// ---- DUTs/IO/Boxes/KL_65B88BEE.TcDUT
{attribute 'GeneratedUsingTerminal: KL1862-0001'}
{attribute addProperty BoxType "KL1862-0001"}
{attribute addProperty Description ""}
{attribute addProperty Physics ""}
{attribute addProperty Id "Channel_1AT %I*Channel_87C95E760Channel_2AT %I*Channel_87C95E760Channel_3AT %I*Channel_87C95E760Channel_4AT %I*Channel_87C95E760Channel_5AT %I*Channel_87C95E760Channel_6AT %I*Channel_87C95E760Channel_7AT %I*Channel_87C95E760Channel_8AT %I*Channel_87C95E760Channel_9AT %I*Channel_87C95E760Channel_10AT %I*Channel_87C95E760Channel_11AT %I*Channel_87C95E760Channel_12AT %I*Channel_87C95E760Channel_13AT %I*Channel_87C95E760Channel_14AT %I*Channel_87C95E760Channel_15AT %I*Channel_87C95E760Channel_16AT %I*Channel_87C95E760"}
{attribute addProperty CRC "1706593262"}
{attribute addProperty Size "0"}
TYPE KL_65B88BEE :
STRUCT
	{attribute addProperty Name "Channel_1"}
	Channel_1 : Channel_87C95E76;
	{attribute addProperty Name "Channel_2"}
	Channel_2 : Channel_87C95E76;
	{attribute addProperty Name "Channel_3"}
	Channel_3 : Channel_87C95E76;
	{attribute addProperty Name "Channel_4"}
	Channel_4 : Channel_87C95E76;
	{attribute addProperty Name "Channel_5"}
	Channel_5 : Channel_87C95E76;
	{attribute addProperty Name "Channel_6"}
	Channel_6 : Channel_87C95E76;
	{attribute addProperty Name "Channel_7"}
	Channel_7 : Channel_87C95E76;
	{attribute addProperty Name "Channel_8"}
	Channel_8 : Channel_87C95E76;
	{attribute addProperty Name "Channel_9"}
	Channel_9 : Channel_87C95E76;
	{attribute addProperty Name "Channel_10"}
	Channel_10 : Channel_87C95E76;
	{attribute addProperty Name "Channel_11"}
	Channel_11 : Channel_87C95E76;
	{attribute addProperty Name "Channel_12"}
	Channel_12 : Channel_87C95E76;
	{attribute addProperty Name "Channel_13"}
	Channel_13 : Channel_87C95E76;
	{attribute addProperty Name "Channel_14"}
	Channel_14 : Channel_87C95E76;
	{attribute addProperty Name "Channel_15"}
	Channel_15 : Channel_87C95E76;
	{attribute addProperty Name "Channel_16"}
	Channel_16 : Channel_87C95E76;
END_STRUCT
END_TYPE

// ---- DUTs/IO/Boxes/KL1872_65B88BEE.TcDUT
{attribute 'GeneratedUsingTerminal: KL1872'}
{attribute addProperty BoxType "KL1872"}
{attribute addProperty Description ""}
{attribute addProperty Physics ""}
{attribute addProperty Id "Channel_1AT %I*Channel_87C95E760Channel_2AT %I*Channel_87C95E760Channel_3AT %I*Channel_87C95E760Channel_4AT %I*Channel_87C95E760Channel_5AT %I*Channel_87C95E760Channel_6AT %I*Channel_87C95E760Channel_7AT %I*Channel_87C95E760Channel_8AT %I*Channel_87C95E760Channel_9AT %I*Channel_87C95E760Channel_10AT %I*Channel_87C95E760Channel_11AT %I*Channel_87C95E760Channel_12AT %I*Channel_87C95E760Channel_13AT %I*Channel_87C95E760Channel_14AT %I*Channel_87C95E760Channel_15AT %I*Channel_87C95E760Channel_16AT %I*Channel_87C95E760"}
{attribute addProperty CRC "1706593262"}
{attribute addProperty Size "0"}
TYPE KL1872_65B88BEE :
STRUCT
	{attribute addProperty Name "Channel_1"}
	Channel_1 : Channel_87C95E76;
	{attribute addProperty Name "Channel_2"}
	Channel_2 : Channel_87C95E76;
	{attribute addProperty Name "Channel_3"}
	Channel_3 : Channel_87C95E76;
	{attribute addProperty Name "Channel_4"}
	Channel_4 : Channel_87C95E76;
	{attribute addProperty Name "Channel_5"}
	Channel_5 : Channel_87C95E76;
	{attribute addProperty Name "Channel_6"}
	Channel_6 : Channel_87C95E76;
	{attribute addProperty Name "Channel_7"}
	Channel_7 : Channel_87C95E76;
	{attribute addProperty Name "Channel_8"}
	Channel_8 : Channel_87C95E76;
	{attribute addProperty Name "Channel_9"}
	Channel_9 : Channel_87C95E76;
	{attribute addProperty Name "Channel_10"}
	Channel_10 : Channel_87C95E76;
	{attribute addProperty Name "Channel_11"}
	Channel_11 : Channel_87C95E76;
	{attribute addProperty Name "Channel_12"}
	Channel_12 : Channel_87C95E76;
	{attribute addProperty Name "Channel_13"}
	Channel_13 : Channel_87C95E76;
	{attribute addProperty Name "Channel_14"}
	Channel_14 : Channel_87C95E76;
	{attribute addProperty Name "Channel_15"}
	Channel_15 : Channel_87C95E76;
	{attribute addProperty Name "Channel_16"}
	Channel_16 : Channel_87C95E76;
END_STRUCT
END_TYPE

// ---- DUTs/IO/Boxes/KL1889_65B88BEE.TcDUT
{attribute 'GeneratedUsingTerminal: KL1889'}
{attribute addProperty BoxType "KL1889"}
{attribute addProperty Description ""}
{attribute addProperty Physics ""}
{attribute addProperty Id "Channel_1AT %I*Channel_87C95E760Channel_2AT %I*Channel_87C95E760Channel_3AT %I*Channel_87C95E760Channel_4AT %I*Channel_87C95E760Channel_5AT %I*Channel_87C95E760Channel_6AT %I*Channel_87C95E760Channel_7AT %I*Channel_87C95E760Channel_8AT %I*Channel_87C95E760Channel_9AT %I*Channel_87C95E760Channel_10AT %I*Channel_87C95E760Channel_11AT %I*Channel_87C95E760Channel_12AT %I*Channel_87C95E760Channel_13AT %I*Channel_87C95E760Channel_14AT %I*Channel_87C95E760Channel_15AT %I*Channel_87C95E760Channel_16AT %I*Channel_87C95E760"}
{attribute addProperty CRC "1706593262"}
{attribute addProperty Size "0"}
TYPE KL1889_65B88BEE :
STRUCT
	{attribute addProperty Name "Channel_1"}
	Channel_1 : Channel_87C95E76;
	{attribute addProperty Name "Channel_2"}
	Channel_2 : Channel_87C95E76;
	{attribute addProperty Name "Channel_3"}
	Channel_3 : Channel_87C95E76;
	{attribute addProperty Name "Channel_4"}
	Channel_4 : Channel_87C95E76;
	{attribute addProperty Name "Channel_5"}
	Channel_5 : Channel_87C95E76;
	{attribute addProperty Name "Channel_6"}
	Channel_6 : Channel_87C95E76;
	{attribute addProperty Name "Channel_7"}
	Channel_7 : Channel_87C95E76;
	{attribute addProperty Name "Channel_8"}
	Channel_8 : Channel_87C95E76;
	{attribute addProperty Name "Channel_9"}
	Channel_9 : Channel_87C95E76;
	{attribute addProperty Name "Channel_10"}
	Channel_10 : Channel_87C95E76;
	{attribute addProperty Name "Channel_11"}
	Channel_11 : Channel_87C95E76;
	{attribute addProperty Name "Channel_12"}
	Channel_12 : Channel_87C95E76;
	{attribute addProperty Name "Channel_13"}
	Channel_13 : Channel_87C95E76;
	{attribute addProperty Name "Channel_14"}
	Channel_14 : Channel_87C95E76;
	{attribute addProperty Name "Channel_15"}
	Channel_15 : Channel_87C95E76;
	{attribute addProperty Name "Channel_16"}
	Channel_16 : Channel_87C95E76;
END_STRUCT
END_TYPE

// ---- DUTs/IO/Boxes/KL1904_7F0D69A9.TcDUT
{attribute 'GeneratedUsingTerminal: KL1904'}
{attribute addProperty BoxType "KL1904"}
{attribute addProperty Description ""}
{attribute addProperty Physics ""}
{attribute addProperty Id "Channel_1AT %Q*Channel_1D6668A90"}
{attribute addProperty CRC "2131585449"}
{attribute addProperty Size "0"}
TYPE KL1904_7F0D69A9 :
STRUCT
	{attribute addProperty Name "Channel_1"}
	Channel_1 : Channel_1D6668A9;
END_STRUCT
END_TYPE

// ---- DUTs/IO/Boxes/KL1908_7F0D69A9.TcDUT
{attribute 'GeneratedUsingTerminal: KL1908'}
{attribute addProperty BoxType "KL1908"}
{attribute addProperty Description ""}
{attribute addProperty Physics ""}
{attribute addProperty Id "Channel_1AT %Q*Channel_1D6668A90"}
{attribute addProperty CRC "2131585449"}
{attribute addProperty Size "0"}
TYPE KL1908_7F0D69A9 :
STRUCT
	{attribute addProperty Name "Channel_1"}
	Channel_1 : Channel_1D6668A9;
END_STRUCT
END_TYPE

// ---- DUTs/IO/Boxes/KL_ABE34026.TcDUT
{attribute 'GeneratedUsingTerminal: KL1004-0050'}
{attribute addProperty BoxType "KL1004-0050"}
{attribute addProperty Description ""}
{attribute addProperty Physics ""}
{attribute addProperty Id "Channel_1AT %I*Channel_87C95E760Channel_2AT %I*Channel_87C95E760Channel_3AT %I*Channel_87C95E760Channel_4AT %I*Channel_87C95E760Channel_5AT %I*Channel_87C95E760Channel_6AT %I*Channel_87C95E760Channel_7AT %I*Channel_87C95E760Channel_8AT %I*Channel_87C95E760Channel_9AT %I*Channel_87C95E760Channel_10AT %I*Channel_87C95E760Channel_11AT %I*Channel_87C95E760Channel_12AT %I*Channel_87C95E760Channel_13AT %I*Channel_87C95E760Channel_14AT %I*Channel_87C95E760Channel_15AT %I*Channel_87C95E760Channel_16AT %I*Channel_87C95E760Channel_17AT %I*Channel_87C95E760Channel_18AT %I*Channel_87C95E760Channel_19AT %I*Channel_87C95E760Channel_20AT %I*Channel_87C95E760Channel_21AT %I*Channel_87C95E760Channel_22AT %I*Channel_87C95E760Channel_23AT %I*Channel_87C95E760Channel_24AT %I*Channel_87C95E760Channel_25AT %I*Channel_87C95E760Channel_26AT %I*Channel_87C95E760Channel_27AT %I*Channel_87C95E760Channel_28AT %I*Channel_87C95E760Channel_29AT %I*Channel_87C95E760Channel_30AT %I*Channel_87C95E760Channel_31AT %I*Channel_87C95E760Channel_32AT %I*Channel_87C95E760"}
{attribute addProperty CRC "2883797030"}
{attribute addProperty Size "0"}
TYPE KL_ABE34026 :
STRUCT
	{attribute addProperty Name "Channel_1"}
	Channel_1 : Channel_87C95E76;
	{attribute addProperty Name "Channel_2"}
	Channel_2 : Channel_87C95E76;
	{attribute addProperty Name "Channel_3"}
	Channel_3 : Channel_87C95E76;
	{attribute addProperty Name "Channel_4"}
	Channel_4 : Channel_87C95E76;
	{attribute addProperty Name "Channel_5"}
	Channel_5 : Channel_87C95E76;
	{attribute addProperty Name "Channel_6"}
	Channel_6 : Channel_87C95E76;
	{attribute addProperty Name "Channel_7"}
	Channel_7 : Channel_87C95E76;
	{attribute addProperty Name "Channel_8"}
	Channel_8 : Channel_87C95E76;
	{attribute addProperty Name "Channel_9"}
	Channel_9 : Channel_87C95E76;
	{attribute addProperty Name "Channel_10"}
	Channel_10 : Channel_87C95E76;
	{attribute addProperty Name "Channel_11"}
	Channel_11 : Channel_87C95E76;
	{attribute addProperty Name "Channel_12"}
	Channel_12 : Channel_87C95E76;
	{attribute addProperty Name "Channel_13"}
	Channel_13 : Channel_87C95E76;
	{attribute addProperty Name "Channel_14"}
	Channel_14 : Channel_87C95E76;
	{attribute addProperty Name "Channel_15"}
	Channel_15 : Channel_87C95E76;
	{attribute addProperty Name "Channel_16"}
	Channel_16 : Channel_87C95E76;
	{attribute addProperty Name "Channel_17"}
	Channel_17 : Channel_87C95E76;
	{attribute addProperty Name "Channel_18"}
	Channel_18 : Channel_87C95E76;
	{attribute addProperty Name "Channel_19"}
	Channel_19 : Channel_87C95E76;
	{attribute addProperty Name "Channel_20"}
	Channel_20 : Channel_87C95E76;
	{attribute addProperty Name "Channel_21"}
	Channel_21 : Channel_87C95E76;
	{attribute addProperty Name "Channel_22"}
	Channel_22 : Channel_87C95E76;
	{attribute addProperty Name "Channel_23"}
	Channel_23 : Channel_87C95E76;
	{attribute addProperty Name "Channel_24"}
	Channel_24 : Channel_87C95E76;
	{attribute addProperty Name "Channel_25"}
	Channel_25 : Channel_87C95E76;
	{attribute addProperty Name "Channel_26"}
	Channel_26 : Channel_87C95E76;
	{attribute addProperty Name "Channel_27"}
	Channel_27 : Channel_87C95E76;
	{attribute addProperty Name "Channel_28"}
	Channel_28 : Channel_87C95E76;
	{attribute addProperty Name "Channel_29"}
	Channel_29 : Channel_87C95E76;
	{attribute addProperty Name "Channel_30"}
	Channel_30 : Channel_87C95E76;
	{attribute addProperty Name "Channel_31"}
	Channel_31 : Channel_87C95E76;
	{attribute addProperty Name "Channel_32"}
	Channel_32 : Channel_87C95E76;
END_STRUCT
END_TYPE

// ---- DUTs/IO/Boxes/KL_E882B8F1.TcDUT
{attribute 'GeneratedUsingTerminal: KL1008-0050'}
{attribute addProperty BoxType "KL1008-0050"}
{attribute addProperty Description ""}
{attribute addProperty Physics ""}
{attribute addProperty Id "Channel_1AT %I*Channel_87C95E760Channel_2AT %I*Channel_87C95E760Channel_3AT %I*Channel_87C95E760Channel_4AT %I*Channel_87C95E760Channel_5AT %I*Channel_87C95E760Channel_6AT %I*Channel_87C95E760Channel_7AT %I*Channel_87C95E760Channel_8AT %I*Channel_87C95E760Channel_9AT %I*Channel_87C95E760Channel_10AT %I*Channel_87C95E760Channel_11AT %I*Channel_87C95E760Channel_12AT %I*Channel_87C95E760Channel_13AT %I*Channel_87C95E760Channel_14AT %I*Channel_87C95E760Channel_15AT %I*Channel_87C95E760Channel_16AT %I*Channel_87C95E760Channel_17AT %I*Channel_87C95E760Channel_18AT %I*Channel_87C95E760Channel_19AT %I*Channel_87C95E760Channel_20AT %I*Channel_87C95E760Channel_21AT %I*Channel_87C95E760Channel_22AT %I*Channel_87C95E760Channel_23AT %I*Channel_87C95E760Channel_24AT %I*Channel_87C95E760Channel_25AT %I*Channel_87C95E760Channel_26AT %I*Channel_87C95E760Channel_27AT %I*Channel_87C95E760Channel_28AT %I*Channel_87C95E760Channel_29AT %I*Channel_87C95E760Channel_30AT %I*Channel_87C95E760Channel_31AT %I*Channel_87C95E760Channel_32AT %I*Channel_87C95E760Channel_33AT %I*Channel_87C95E760Channel_34AT %I*Channel_87C95E760Channel_35AT %I*Channel_87C95E760Channel_36AT %I*Channel_87C95E760Channel_37AT %I*Channel_87C95E760Channel_38AT %I*Channel_87C95E760Channel_39AT %I*Channel_87C95E760Channel_40AT %I*Channel_87C95E760Channel_41AT %I*Channel_87C95E760Channel_42AT %I*Channel_87C95E760Channel_43AT %I*Channel_87C95E760Channel_44AT %I*Channel_87C95E760Channel_45AT %I*Channel_87C95E760Channel_46AT %I*Channel_87C95E760Channel_47AT %I*Channel_87C95E760Channel_48AT %I*Channel_87C95E760Channel_49AT %I*Channel_87C95E760Channel_50AT %I*Channel_87C95E760Channel_51AT %I*Channel_87C95E760Channel_52AT %I*Channel_87C95E760Channel_53AT %I*Channel_87C95E760Channel_54AT %I*Channel_87C95E760Channel_55AT %I*Channel_87C95E760Channel_56AT %I*Channel_87C95E760Channel_57AT %I*Channel_87C95E760Channel_58AT %I*Channel_87C95E760Channel_59AT %I*Channel_87C95E760Channel_60AT %I*Channel_87C95E760Channel_61AT %I*Channel_87C95E760Channel_62AT %I*Channel_87C95E760Channel_63AT %I*Channel_87C95E760Channel_64AT %I*Channel_87C95E760"}
{attribute addProperty CRC "3900881137"}
{attribute addProperty Size "0"}
TYPE KL_E882B8F1 :
STRUCT
	{attribute addProperty Name "Channel_1"}
	Channel_1 : Channel_87C95E76;
	{attribute addProperty Name "Channel_2"}
	Channel_2 : Channel_87C95E76;
	{attribute addProperty Name "Channel_3"}
	Channel_3 : Channel_87C95E76;
	{attribute addProperty Name "Channel_4"}
	Channel_4 : Channel_87C95E76;
	{attribute addProperty Name "Channel_5"}
	Channel_5 : Channel_87C95E76;
	{attribute addProperty Name "Channel_6"}
	Channel_6 : Channel_87C95E76;
	{attribute addProperty Name "Channel_7"}
	Channel_7 : Channel_87C95E76;
	{attribute addProperty Name "Channel_8"}
	Channel_8 : Channel_87C95E76;
	{attribute addProperty Name "Channel_9"}
	Channel_9 : Channel_87C95E76;
	{attribute addProperty Name "Channel_10"}
	Channel_10 : Channel_87C95E76;
	{attribute addProperty Name "Channel_11"}
	Channel_11 : Channel_87C95E76;
	{attribute addProperty Name "Channel_12"}
	Channel_12 : Channel_87C95E76;
	{attribute addProperty Name "Channel_13"}
	Channel_13 : Channel_87C95E76;
	{attribute addProperty Name "Channel_14"}
	Channel_14 : Channel_87C95E76;
	{attribute addProperty Name "Channel_15"}
	Channel_15 : Channel_87C95E76;
	{attribute addProperty Name "Channel_16"}
	Channel_16 : Channel_87C95E76;
	{attribute addProperty Name "Channel_17"}
	Channel_17 : Channel_87C95E76;
	{attribute addProperty Name "Channel_18"}
	Channel_18 : Channel_87C95E76;
	{attribute addProperty Name "Channel_19"}
	Channel_19 : Channel_87C95E76;
	{attribute addProperty Name "Channel_20"}
	Channel_20 : Channel_87C95E76;
	{attribute addProperty Name "Channel_21"}
	Channel_21 : Channel_87C95E76;
	{attribute addProperty Name "Channel_22"}
	Channel_22 : Channel_87C95E76;
	{attribute addProperty Name "Channel_23"}
	Channel_23 : Channel_87C95E76;
	{attribute addProperty Name "Channel_24"}
	Channel_24 : Channel_87C95E76;
	{attribute addProperty Name "Channel_25"}
	Channel_25 : Channel_87C95E76;
	{attribute addProperty Name "Channel_26"}
	Channel_26 : Channel_87C95E76;
	{attribute addProperty Name "Channel_27"}
	Channel_27 : Channel_87C95E76;
	{attribute addProperty Name "Channel_28"}
	Channel_28 : Channel_87C95E76;
	{attribute addProperty Name "Channel_29"}
	Channel_29 : Channel_87C95E76;
	{attribute addProperty Name "Channel_30"}
	Channel_30 : Channel_87C95E76;
	{attribute addProperty Name "Channel_31"}
	Channel_31 : Channel_87C95E76;
	{attribute addProperty Name "Channel_32"}
	Channel_32 : Channel_87C95E76;
	{attribute addProperty Name "Channel_33"}
	Channel_33 : Channel_87C95E76;
	{attribute addProperty Name "Channel_34"}
	Channel_34 : Channel_87C95E76;
	{attribute addProperty Name "Channel_35"}
	Channel_35 : Channel_87C95E76;
	{attribute addProperty Name "Channel_36"}
	Channel_36 : Channel_87C95E76;
	{attribute addProperty Name "Channel_37"}
	Channel_37 : Channel_87C95E76;
	{attribute addProperty Name "Channel_38"}
	Channel_38 : Channel_87C95E76;
	{attribute addProperty Name "Channel_39"}
	Channel_39 : Channel_87C95E76;
	{attribute addProperty Name "Channel_40"}
	Channel_40 : Channel_87C95E76;
	{attribute addProperty Name "Channel_41"}
	Channel_41 : Channel_87C95E76;
	{attribute addProperty Name "Channel_42"}
	Channel_42 : Channel_87C95E76;
	{attribute addProperty Name "Channel_43"}
	Channel_43 : Channel_87C95E76;
	{attribute addProperty Name "Channel_44"}
	Channel_44 : Channel_87C95E76;
	{attribute addProperty Name "Channel_45"}
	Channel_45 : Channel_87C95E76;
	{attribute addProperty Name "Channel_46"}
	Channel_46 : Channel_87C95E76;
	{attribute addProperty Name "Channel_47"}
	Channel_47 : Channel_87C95E76;
	{attribute addProperty Name "Channel_48"}
	Channel_48 : Channel_87C95E76;
	{attribute addProperty Name "Channel_49"}
	Channel_49 : Channel_87C95E76;
	{attribute addProperty Name "Channel_50"}
	Channel_50 : Channel_87C95E76;
	{attribute addProperty Name "Channel_51"}
	Channel_51 : Channel_87C95E76;
	{attribute addProperty Name "Channel_52"}
	Channel_52 : Channel_87C95E76;
	{attribute addProperty Name "Channel_53"}
	Channel_53 : Channel_87C95E76;
	{attribute addProperty Name "Channel_54"}
	Channel_54 : Channel_87C95E76;
	{attribute addProperty Name "Channel_55"}
	Channel_55 : Channel_87C95E76;
	{attribute addProperty Name "Channel_56"}
	Channel_56 : Channel_87C95E76;
	{attribute addProperty Name "Channel_57"}
	Channel_57 : Channel_87C95E76;
	{attribute addProperty Name "Channel_58"}
	Channel_58 : Channel_87C95E76;
	{attribute addProperty Name "Channel_59"}
	Channel_59 : Channel_87C95E76;
	{attribute addProperty Name "Channel_60"}
	Channel_60 : Channel_87C95E76;
	{attribute addProperty Name "Channel_61"}
	Channel_61 : Channel_87C95E76;
	{attribute addProperty Name "Channel_62"}
	Channel_62 : Channel_87C95E76;
	{attribute addProperty Name "Channel_63"}
	Channel_63 : Channel_87C95E76;
	{attribute addProperty Name "Channel_64"}
	Channel_64 : Channel_87C95E76;
END_STRUCT
END_TYPE

// ---- DUTs/IO/Boxes/KL_52751275.TcDUT
{attribute 'GeneratedUsingTerminal: KL1644-0050'}
{attribute addProperty BoxType "KL1644-0050"}
{attribute addProperty Description ""}
{attribute addProperty Physics ""}
{attribute addProperty Id "Channel_1AT %Q*Channel_6B723A160Channel_2AT %Q*Channel_6B723A160Channel_3AT %Q*Channel_6B723A160Channel_4AT %Q*Channel_6B723A160"}
{attribute addProperty CRC "1383404149"}
{attribute addProperty Size "0"}
TYPE KL_52751275 :
STRUCT
	{attribute addProperty Name "Channel_1"}
	Channel_1 : Channel_6B723A16;
	{attribute addProperty Name "Channel_2"}
	Channel_2 : Channel_6B723A16;
	{attribute addProperty Name "Channel_3"}
	Channel_3 : Channel_6B723A16;
	{attribute addProperty Name "Channel_4"}
	Channel_4 : Channel_6B723A16;
END_STRUCT
END_TYPE

// ---- DUTs/IO/Boxes/KL2012_DCA75612.TcDUT
{attribute 'GeneratedUsingTerminal: KL2012'}
{attribute addProperty BoxType "KL2012"}
{attribute addProperty Description ""}
{attribute addProperty Physics ""}
{attribute addProperty Id "Channel_1AT %Q*Channel_460B8C400Channel_2AT %Q*Channel_460B8C400"}
{attribute addProperty CRC "3701954066"}
{attribute addProperty Size "0"}
TYPE KL2012_DCA75612 :
STRUCT
	{attribute addProperty Name "Channel_1"}
	Channel_1 : Channel_460B8C40;
	{attribute addProperty Name "Channel_2"}
	Channel_2 : Channel_460B8C40;
END_STRUCT
END_TYPE

// ---- DUTs/IO/Boxes/KL2022_DCA75612.TcDUT
{attribute 'GeneratedUsingTerminal: KL2022'}
{attribute addProperty BoxType "KL2022"}
{attribute addProperty Description ""}
{attribute addProperty Physics ""}
{attribute addProperty Id "Channel_1AT %Q*Channel_460B8C400Channel_2AT %Q*Channel_460B8C400"}
{attribute addProperty CRC "3701954066"}
{attribute addProperty Size "0"}
TYPE KL2022_DCA75612 :
STRUCT
	{attribute addProperty Name "Channel_1"}
	Channel_1 : Channel_460B8C40;
	{attribute addProperty Name "Channel_2"}
	Channel_2 : Channel_460B8C40;
END_STRUCT
END_TYPE

// ---- DUTs/IO/Boxes/KL2032_DCA75612.TcDUT
{attribute 'GeneratedUsingTerminal: KL2032'}
{attribute addProperty BoxType "KL2032"}
{attribute addProperty Description ""}
{attribute addProperty Physics ""}
{attribute addProperty Id "Channel_1AT %Q*Channel_460B8C400Channel_2AT %Q*Channel_460B8C400"}
{attribute addProperty CRC "3701954066"}
{attribute addProperty Size "0"}
TYPE KL2032_DCA75612 :
STRUCT
	{attribute addProperty Name "Channel_1"}
	Channel_1 : Channel_460B8C40;
	{attribute addProperty Name "Channel_2"}
	Channel_2 : Channel_460B8C40;
END_STRUCT
END_TYPE

// ---- DUTs/IO/Boxes/KL2114_E49EE1EF.TcDUT
{attribute 'GeneratedUsingTerminal: KL2114'}
{attribute addProperty BoxType "KL2114"}
{attribute addProperty Description ""}
{attribute addProperty Physics ""}
{attribute addProperty Id "Channel_1AT %Q*Channel_460B8C400Channel_2AT %Q*Channel_460B8C400Channel_3AT %Q*Channel_460B8C400Channel_4AT %Q*Channel_460B8C400"}
{attribute addProperty CRC "3835617775"}
{attribute addProperty Size "0"}
TYPE KL2114_E49EE1EF :
STRUCT
	{attribute addProperty Name "Channel_1"}
	Channel_1 : Channel_460B8C40;
	{attribute addProperty Name "Channel_2"}
	Channel_2 : Channel_460B8C40;
	{attribute addProperty Name "Channel_3"}
	Channel_3 : Channel_460B8C40;
	{attribute addProperty Name "Channel_4"}
	Channel_4 : Channel_460B8C40;
END_STRUCT
END_TYPE

// ---- DUTs/IO/Boxes/KL2124_E49EE1EF.TcDUT
{attribute 'GeneratedUsingTerminal: KL2124'}
{attribute addProperty BoxType "KL2124"}
{attribute addProperty Description ""}
{attribute addProperty Physics ""}
{attribute addProperty Id "Channel_1AT %Q*Channel_460B8C400Channel_2AT %Q*Channel_460B8C400Channel_3AT %Q*Channel_460B8C400Channel_4AT %Q*Channel_460B8C400"}
{attribute addProperty CRC "3835617775"}
{attribute addProperty Size "0"}
TYPE KL2124_E49EE1EF :
STRUCT
	{attribute addProperty Name "Channel_1"}
	Channel_1 : Channel_460B8C40;
	{attribute addProperty Name "Channel_2"}
	Channel_2 : Channel_460B8C40;
	{attribute addProperty Name "Channel_3"}
	Channel_3 : Channel_460B8C40;
	{attribute addProperty Name "Channel_4"}
	Channel_4 : Channel_460B8C40;
END_STRUCT
END_TYPE

// ---- DUTs/IO/Boxes/KL2134_E49EE1EF.TcDUT
{attribute 'GeneratedUsingTerminal: KL2134'}
{attribute addProperty BoxType "KL2134"}
{attribute addProperty Description ""}
{attribute addProperty Physics ""}
{attribute addProperty Id "Channel_1AT %Q*Channel_460B8C400Channel_2AT %Q*Channel_460B8C400Channel_3AT %Q*Channel_460B8C400Channel_4AT %Q*Channel_460B8C400"}
{attribute addProperty CRC "3835617775"}
{attribute addProperty Size "0"}
TYPE KL2134_E49EE1EF :
STRUCT
	{attribute addProperty Name "Channel_1"}
	Channel_1 : Channel_460B8C40;
	{attribute addProperty Name "Channel_2"}
	Channel_2 : Channel_460B8C40;
	{attribute addProperty Name "Channel_3"}
	Channel_3 : Channel_460B8C40;
	{attribute addProperty Name "Channel_4"}
	Channel_4 : Channel_460B8C40;
END_STRUCT
END_TYPE

// ---- DUTs/IO/Boxes/KL2184_E49EE1EF.TcDUT
{attribute 'GeneratedUsingTerminal: KL2184'}
{attribute addProperty BoxType "KL2184"}
{attribute addProperty Description ""}
{attribute addProperty Physics ""}
{attribute addProperty Id "Channel_1AT %Q*Channel_460B8C400Channel_2AT %Q*Channel_460B8C400Channel_3AT %Q*Channel_460B8C400Channel_4AT %Q*Channel_460B8C400"}
{attribute addProperty CRC "3835617775"}
{attribute addProperty Size "0"}
TYPE KL2184_E49EE1EF :
STRUCT
	{attribute addProperty Name "Channel_1"}
	Channel_1 : Channel_460B8C40;
	{attribute addProperty Name "Channel_2"}
	Channel_2 : Channel_460B8C40;
	{attribute addProperty Name "Channel_3"}
	Channel_3 : Channel_460B8C40;
	{attribute addProperty Name "Channel_4"}
	Channel_4 : Channel_460B8C40;
END_STRUCT
END_TYPE

// ---- DUTs/IO/Boxes/KL2212_BA18203A.TcDUT
{attribute 'GeneratedUsingTerminal: KL2212'}
{attribute addProperty BoxType "KL2212"}
{attribute addProperty Description ""}
{attribute addProperty Physics ""}
{attribute addProperty Id "Channel_1AT %Q*Channel_DCF170BB0Channel_2AT %Q*Channel_DCF170BB0"}
{attribute addProperty CRC "3122143290"}
{attribute addProperty Size "0"}
TYPE KL2212_BA18203A :
STRUCT
	{attribute addProperty Name "Channel_1"}
	Channel_1 : Channel_DCF170BB;
	{attribute addProperty Name "Channel_2"}
	Channel_2 : Channel_DCF170BB;
END_STRUCT
END_TYPE

// ---- DUTs/IO/Boxes/KL1202_EC84F46C.TcDUT
{attribute 'GeneratedUsingTerminal: KL1202'}
{attribute addProperty BoxType "KL1202"}
{attribute addProperty Description ""}
{attribute addProperty Physics ""}
{attribute addProperty Id "Channel_1AT %Q*Channel_72DF63360Channel_2AT %Q*Channel_72DF63360"}
{attribute addProperty CRC "3968136300"}
{attribute addProperty Size "0"}
TYPE KL1202_EC84F46C :
STRUCT
	{attribute addProperty Name "Channel_1"}
	Channel_1 : Channel_72DF6336;
	{attribute addProperty Name "Channel_2"}
	Channel_2 : Channel_72DF6336;
END_STRUCT
END_TYPE

// ---- DUTs/IO/Boxes/KL2404_E49EE1EF.TcDUT
{attribute 'GeneratedUsingTerminal: KL2404'}
{attribute addProperty BoxType "KL2404"}
{attribute addProperty Description ""}
{attribute addProperty Physics ""}
{attribute addProperty Id "Channel_1AT %Q*Channel_460B8C400Channel_2AT %Q*Channel_460B8C400Channel_3AT %Q*Channel_460B8C400Channel_4AT %Q*Channel_460B8C400"}
{attribute addProperty CRC "3835617775"}
{attribute addProperty Size "0"}
TYPE KL2404_E49EE1EF :
STRUCT
	{attribute addProperty Name "Channel_1"}
	Channel_1 : Channel_460B8C40;
	{attribute addProperty Name "Channel_2"}
	Channel_2 : Channel_460B8C40;
	{attribute addProperty Name "Channel_3"}
	Channel_3 : Channel_460B8C40;
	{attribute addProperty Name "Channel_4"}
	Channel_4 : Channel_460B8C40;
END_STRUCT
END_TYPE

// ---- DUTs/IO/Boxes/KL2408_CBAD53BF.TcDUT
{attribute 'GeneratedUsingTerminal: KL2408'}
{attribute addProperty BoxType "KL2408"}
{attribute addProperty Description ""}
{attribute addProperty Physics ""}
{attribute addProperty Id "Channel_1AT %Q*Channel_460B8C400Channel_2AT %Q*Channel_460B8C400Channel_3AT %Q*Channel_460B8C400Channel_4AT %Q*Channel_460B8C400Channel_5AT %Q*Channel_460B8C400Channel_6AT %Q*Channel_460B8C400Channel_7AT %Q*Channel_460B8C400Channel_8AT %Q*Channel_460B8C400"}
{attribute addProperty CRC "3417134015"}
{attribute addProperty Size "0"}
TYPE KL2408_CBAD53BF :
STRUCT
	{attribute addProperty Name "Channel_1"}
	Channel_1 : Channel_460B8C40;
	{attribute addProperty Name "Channel_2"}
	Channel_2 : Channel_460B8C40;
	{attribute addProperty Name "Channel_3"}
	Channel_3 : Channel_460B8C40;
	{attribute addProperty Name "Channel_4"}
	Channel_4 : Channel_460B8C40;
	{attribute addProperty Name "Channel_5"}
	Channel_5 : Channel_460B8C40;
	{attribute addProperty Name "Channel_6"}
	Channel_6 : Channel_460B8C40;
	{attribute addProperty Name "Channel_7"}
	Channel_7 : Channel_460B8C40;
	{attribute addProperty Name "Channel_8"}
	Channel_8 : Channel_460B8C40;
END_STRUCT
END_TYPE

// ---- DUTs/IO/Boxes/KL2424_E49EE1EF.TcDUT
{attribute 'GeneratedUsingTerminal: KL2424'}
{attribute addProperty BoxType "KL2424"}
{attribute addProperty Description ""}
{attribute addProperty Physics ""}
{attribute addProperty Id "Channel_1AT %Q*Channel_460B8C400Channel_2AT %Q*Channel_460B8C400Channel_3AT %Q*Channel_460B8C400Channel_4AT %Q*Channel_460B8C400"}
{attribute addProperty CRC "3835617775"}
{attribute addProperty Size "0"}
TYPE KL2424_E49EE1EF :
STRUCT
	{attribute addProperty Name "Channel_1"}
	Channel_1 : Channel_460B8C40;
	{attribute addProperty Name "Channel_2"}
	Channel_2 : Channel_460B8C40;
	{attribute addProperty Name "Channel_3"}
	Channel_3 : Channel_460B8C40;
	{attribute addProperty Name "Channel_4"}
	Channel_4 : Channel_460B8C40;
END_STRUCT
END_TYPE

// ---- DUTs/IO/Boxes/KL2442_DCA75612.TcDUT
{attribute 'GeneratedUsingTerminal: KL2442'}
{attribute addProperty BoxType "KL2442"}
{attribute addProperty Description ""}
{attribute addProperty Physics ""}
{attribute addProperty Id "Channel_1AT %Q*Channel_460B8C400Channel_2AT %Q*Channel_460B8C400"}
{attribute addProperty CRC "3701954066"}
{attribute addProperty Size "0"}
TYPE KL2442_DCA75612 :
STRUCT
	{attribute addProperty Name "Channel_1"}
	Channel_1 : Channel_460B8C40;
	{attribute addProperty Name "Channel_2"}
	Channel_2 : Channel_460B8C40;
END_STRUCT
END_TYPE

// ---- DUTs/IO/Boxes/KL2488_CBAD53BF.TcDUT
{attribute 'GeneratedUsingTerminal: KL2488'}
{attribute addProperty BoxType "KL2488"}
{attribute addProperty Description ""}
{attribute addProperty Physics ""}
{attribute addProperty Id "Channel_1AT %Q*Channel_460B8C400Channel_2AT %Q*Channel_460B8C400Channel_3AT %Q*Channel_460B8C400Channel_4AT %Q*Channel_460B8C400Channel_5AT %Q*Channel_460B8C400Channel_6AT %Q*Channel_460B8C400Channel_7AT %Q*Channel_460B8C400Channel_8AT %Q*Channel_460B8C400"}
{attribute addProperty CRC "3417134015"}
{attribute addProperty Size "0"}
TYPE KL2488_CBAD53BF :
STRUCT
	{attribute addProperty Name "Channel_1"}
	Channel_1 : Channel_460B8C40;
	{attribute addProperty Name "Channel_2"}
	Channel_2 : Channel_460B8C40;
	{attribute addProperty Name "Channel_3"}
	Channel_3 : Channel_460B8C40;
	{attribute addProperty Name "Channel_4"}
	Channel_4 : Channel_460B8C40;
	{attribute addProperty Name "Channel_5"}
	Channel_5 : Channel_460B8C40;
	{attribute addProperty Name "Channel_6"}
	Channel_6 : Channel_460B8C40;
	{attribute addProperty Name "Channel_7"}
	Channel_7 : Channel_460B8C40;
	{attribute addProperty Name "Channel_8"}
	Channel_8 : Channel_460B8C40;
END_STRUCT
END_TYPE

// ---- DUTs/IO/Boxes/KL2284_008A18FD.TcDUT
{attribute 'GeneratedUsingTerminal: KL2284'}
{attribute addProperty BoxType "KL2284"}
{attribute addProperty Description ""}
{attribute addProperty Physics ""}
{attribute addProperty Id "Channel_1AT %Q*Channel_26FC8FD80Channel_2AT %Q*Channel_26FC8FD80Channel_3AT %Q*Channel_26FC8FD80Channel_4AT %Q*Channel_26FC8FD80"}
{attribute addProperty CRC "9050365"}
{attribute addProperty Size "0"}
TYPE KL2284_008A18FD :
STRUCT
	{attribute addProperty Name "Channel_1"}
	Channel_1 : Channel_26FC8FD8;
	{attribute addProperty Name "Channel_2"}
	Channel_2 : Channel_26FC8FD8;
	{attribute addProperty Name "Channel_3"}
	Channel_3 : Channel_26FC8FD8;
	{attribute addProperty Name "Channel_4"}
	Channel_4 : Channel_26FC8FD8;
END_STRUCT
END_TYPE

// ---- DUTs/IO/Boxes/KL2502_78388DBB.TcDUT
{attribute 'GeneratedUsingTerminal: KL2502'}
{attribute addProperty BoxType "KL2502"}
{attribute addProperty Description ""}
{attribute addProperty Physics ""}
{attribute addProperty Id "Channel_1AT %Q*Channel_03CEAA5E0Channel_2AT %Q*Channel_03CEAA5E0"}
{attribute addProperty CRC "2016972219"}
{attribute addProperty Size "0"}
TYPE KL2502_78388DBB :
STRUCT
	{attribute addProperty Name "Channel_1"}
	Channel_1 : Channel_03CEAA5E;
	{attribute addProperty Name "Channel_2"}
	Channel_2 : Channel_03CEAA5E;
END_STRUCT
END_TYPE

// ---- DUTs/IO/Boxes/KL2512_78388DBB.TcDUT
{attribute 'GeneratedUsingTerminal: KL2512'}
{attribute addProperty BoxType "KL2512"}
{attribute addProperty Description ""}
{attribute addProperty Physics ""}
{attribute addProperty Id "Channel_1AT %Q*Channel_03CEAA5E0Channel_2AT %Q*Channel_03CEAA5E0"}
{attribute addProperty CRC "2016972219"}
{attribute addProperty Size "0"}
TYPE KL2512_78388DBB :
STRUCT
	{attribute addProperty Name "Channel_1"}
	Channel_1 : Channel_03CEAA5E;
	{attribute addProperty Name "Channel_2"}
	Channel_2 : Channel_03CEAA5E;
END_STRUCT
END_TYPE

// ---- DUTs/IO/Boxes/KL2521_D5F34107.TcDUT
{attribute 'GeneratedUsingTerminal: KL2521'}
{attribute addProperty BoxType "KL2521"}
{attribute addProperty Description ""}
{attribute addProperty Physics ""}
{attribute addProperty Id "Channel_1AT %Q*Channel_03CEAA5E0"}
{attribute addProperty CRC "3589488903"}
{attribute addProperty Size "0"}
TYPE KL2521_D5F34107 :
STRUCT
	{attribute addProperty Name "Channel_1"}
	Channel_1 : Channel_03CEAA5E;
END_STRUCT
END_TYPE

// ---- DUTs/IO/Boxes/KL2531_D5AE5504.TcDUT
{attribute 'GeneratedUsingTerminal: KL2531'}
{attribute addProperty BoxType "KL2531"}
{attribute addProperty Description ""}
{attribute addProperty Physics ""}
{attribute addProperty Id "Channel_1AT %Q*Channel_FEA3DBF80"}
{attribute addProperty CRC "3584972036"}
{attribute addProperty Size "0"}
TYPE KL2531_D5AE5504 :
STRUCT
	{attribute addProperty Name "Channel_1"}
	Channel_1 : Channel_FEA3DBF8;
END_STRUCT
END_TYPE

// ---- DUTs/IO/Boxes/KL_5C335388.TcDUT
{attribute 'GeneratedUsingTerminal: KL2531-0001'}
{attribute addProperty BoxType "KL2531-0001"}
{attribute addProperty Description ""}
{attribute addProperty Physics ""}
{attribute addProperty Id "Channel_1AT %Q*Channel_0D1929F00"}
{attribute addProperty CRC "1546867592"}
{attribute addProperty Size "0"}
TYPE KL_5C335388 :
STRUCT
	{attribute addProperty Name "Channel_1"}
	Channel_1 : Channel_0D1929F0;
END_STRUCT
END_TYPE

// ---- DUTs/IO/Boxes/KL2532_B0461874.TcDUT
{attribute 'GeneratedUsingTerminal: KL2532'}
{attribute addProperty BoxType "KL2532"}
{attribute addProperty Description ""}
{attribute addProperty Physics ""}
{attribute addProperty Id "Channel_1AT %Q*Channel_6576A6810Channel_2AT %Q*Channel_6576A6810"}
{attribute addProperty CRC "2957383796"}
{attribute addProperty Size "0"}
TYPE KL2532_B0461874 :
STRUCT
	{attribute addProperty Name "Channel_1"}
	Channel_1 : Channel_6576A681;
	{attribute addProperty Name "Channel_2"}
	Channel_2 : Channel_6576A681;
END_STRUCT
END_TYPE

// ---- DUTs/IO/Boxes/KL2535_B0461874.TcDUT
{attribute 'GeneratedUsingTerminal: KL2535'}
{attribute addProperty BoxType "KL2535"}
{attribute addProperty Description ""}
{attribute addProperty Physics ""}
{attribute addProperty Id "Channel_1AT %Q*Channel_6576A6810Channel_2AT %Q*Channel_6576A6810"}
{attribute addProperty CRC "2957383796"}
{attribute addProperty Size "0"}
TYPE KL2535_B0461874 :
STRUCT
	{attribute addProperty Name "Channel_1"}
	Channel_1 : Channel_6576A681;
	{attribute addProperty Name "Channel_2"}
	Channel_2 : Channel_6576A681;
END_STRUCT
END_TYPE

// ---- DUTs/IO/Boxes/KL_501418F2.TcDUT
{attribute 'GeneratedUsingTerminal: KL2535-0001'}
{attribute addProperty BoxType "KL2535-0001"}
{attribute addProperty Description ""}
{attribute addProperty Physics ""}
{attribute addProperty Id "Channel_1AT %I*0Channel_2AT %I*0"}
{attribute addProperty CRC "1343494386"}
{attribute addProperty Size "0"}
TYPE KL_501418F2 :
STRUCT
	{attribute addProperty Name "Channel_1"}
	Channel_1 : ;
	{attribute addProperty Name "Channel_2"}
	Channel_2 : ;
END_STRUCT
END_TYPE

// ---- DUTs/IO/Boxes/KL2541_D5AE5504.TcDUT
{attribute 'GeneratedUsingTerminal: KL2541'}
{attribute addProperty BoxType "KL2541"}
{attribute addProperty Description ""}
{attribute addProperty Physics ""}
{attribute addProperty Id "Channel_1AT %Q*Channel_FEA3DBF80"}
{attribute addProperty CRC "3584972036"}
{attribute addProperty Size "0"}
TYPE KL2541_D5AE5504 :
STRUCT
	{attribute addProperty Name "Channel_1"}
	Channel_1 : Channel_FEA3DBF8;
END_STRUCT
END_TYPE

// ---- DUTs/IO/Boxes/KL2542_B0461874.TcDUT
{attribute 'GeneratedUsingTerminal: KL2542'}
{attribute addProperty BoxType "KL2542"}
{attribute addProperty Description ""}
{attribute addProperty Physics ""}
{attribute addProperty Id "Channel_1AT %Q*Channel_6576A6810Channel_2AT %Q*Channel_6576A6810"}
{attribute addProperty CRC "2957383796"}
{attribute addProperty Size "0"}
TYPE KL2542_B0461874 :
STRUCT
	{attribute addProperty Name "Channel_1"}
	Channel_1 : Channel_6576A681;
	{attribute addProperty Name "Channel_2"}
	Channel_2 : Channel_6576A681;
END_STRUCT
END_TYPE

// ---- DUTs/IO/Boxes/KL2545_B0461874.TcDUT
{attribute 'GeneratedUsingTerminal: KL2545'}
{attribute addProperty BoxType "KL2545"}
{attribute addProperty Description ""}
{attribute addProperty Physics ""}
{attribute addProperty Id "Channel_1AT %Q*Channel_6576A6810Channel_2AT %Q*Channel_6576A6810"}
{attribute addProperty CRC "2957383796"}
{attribute addProperty Size "0"}
TYPE KL2545_B0461874 :
STRUCT
	{attribute addProperty Name "Channel_1"}
	Channel_1 : Channel_6576A681;
	{attribute addProperty Name "Channel_2"}
	Channel_2 : Channel_6576A681;
END_STRUCT
END_TYPE

// ---- DUTs/IO/Boxes/KL2552_B0461874.TcDUT
{attribute 'GeneratedUsingTerminal: KL2552'}
{attribute addProperty BoxType "KL2552"}
{attribute addProperty Description ""}
{attribute addProperty Physics ""}
{attribute addProperty Id "Channel_1AT %Q*Channel_6576A6810Channel_2AT %Q*Channel_6576A6810"}
{attribute addProperty CRC "2957383796"}
{attribute addProperty Size "0"}
TYPE KL2552_B0461874 :
STRUCT
	{attribute addProperty Name "Channel_1"}
	Channel_1 : Channel_6576A681;
	{attribute addProperty Name "Channel_2"}
	Channel_2 : Channel_6576A681;
END_STRUCT
END_TYPE

// ---- DUTs/IO/Boxes/KL2602_DCA75612.TcDUT
{attribute 'GeneratedUsingTerminal: KL2602'}
{attribute addProperty BoxType "KL2602"}
{attribute addProperty Description ""}
{attribute addProperty Physics ""}
{attribute addProperty Id "Channel_1AT %Q*Channel_460B8C400Channel_2AT %Q*Channel_460B8C400"}
{attribute addProperty CRC "3701954066"}
{attribute addProperty Size "0"}
TYPE KL2602_DCA75612 :
STRUCT
	{attribute addProperty Name "Channel_1"}
	Channel_1 : Channel_460B8C40;
	{attribute addProperty Name "Channel_2"}
	Channel_2 : Channel_460B8C40;
END_STRUCT
END_TYPE

// ---- DUTs/IO/Boxes/KL_DCA75612.TcDUT
{attribute 'GeneratedUsingTerminal: KL2602-0001'}
{attribute addProperty BoxType "KL2602-0001"}
{attribute addProperty Description ""}
{attribute addProperty Physics ""}
{attribute addProperty Id "Channel_1AT %Q*Channel_460B8C400Channel_2AT %Q*Channel_460B8C400"}
{attribute addProperty CRC "3701954066"}
{attribute addProperty Size "0"}
TYPE KL_DCA75612 :
STRUCT
	{attribute addProperty Name "Channel_1"}
	Channel_1 : Channel_460B8C40;
	{attribute addProperty Name "Channel_2"}
	Channel_2 : Channel_460B8C40;
END_STRUCT
END_TYPE

// ---- DUTs/IO/Boxes/KL2612_DCA75612.TcDUT
{attribute 'GeneratedUsingTerminal: KL2612'}
{attribute addProperty BoxType "KL2612"}
{attribute addProperty Description ""}
{attribute addProperty Physics ""}
{attribute addProperty Id "Channel_1AT %Q*Channel_460B8C400Channel_2AT %Q*Channel_460B8C400"}
{attribute addProperty CRC "3701954066"}
{attribute addProperty Size "0"}
TYPE KL2612_DCA75612 :
STRUCT
	{attribute addProperty Name "Channel_1"}
	Channel_1 : Channel_460B8C40;
	{attribute addProperty Name "Channel_2"}
	Channel_2 : Channel_460B8C40;
END_STRUCT
END_TYPE

// ---- DUTs/IO/Boxes/KL2622_DCA75612.TcDUT
{attribute 'GeneratedUsingTerminal: KL2622'}
{attribute addProperty BoxType "KL2622"}
{attribute addProperty Description ""}
{attribute addProperty Physics ""}
{attribute addProperty Id "Channel_1AT %Q*Channel_460B8C400Channel_2AT %Q*Channel_460B8C400"}
{attribute addProperty CRC "3701954066"}
{attribute addProperty Size "0"}
TYPE KL2622_DCA75612 :
STRUCT
	{attribute addProperty Name "Channel_1"}
	Channel_1 : Channel_460B8C40;
	{attribute addProperty Name "Channel_2"}
	Channel_2 : Channel_460B8C40;
END_STRUCT
END_TYPE

// ---- DUTs/IO/Boxes/KL2631_DE78D366.TcDUT
{attribute 'GeneratedUsingTerminal: KL2631'}
{attribute addProperty BoxType "KL2631"}
{attribute addProperty Description ""}
{attribute addProperty Physics ""}
{attribute addProperty Id "Channel_1AT %Q*Channel_460B8C400"}
{attribute addProperty CRC "3732460390"}
{attribute addProperty Size "0"}
TYPE KL2631_DE78D366 :
STRUCT
	{attribute addProperty Name "Channel_1"}
	Channel_1 : Channel_460B8C40;
END_STRUCT
END_TYPE

// ---- DUTs/IO/Boxes/KL2634_E49EE1EF.TcDUT
{attribute 'GeneratedUsingTerminal: KL2634'}
{attribute addProperty BoxType "KL2634"}
{attribute addProperty Description ""}
{attribute addProperty Physics ""}
{attribute addProperty Id "Channel_1AT %Q*Channel_460B8C400Channel_2AT %Q*Channel_460B8C400Channel_3AT %Q*Channel_460B8C400Channel_4AT %Q*Channel_460B8C400"}
{attribute addProperty CRC "3835617775"}
{attribute addProperty Size "0"}
TYPE KL2634_E49EE1EF :
STRUCT
	{attribute addProperty Name "Channel_1"}
	Channel_1 : Channel_460B8C40;
	{attribute addProperty Name "Channel_2"}
	Channel_2 : Channel_460B8C40;
	{attribute addProperty Name "Channel_3"}
	Channel_3 : Channel_460B8C40;
	{attribute addProperty Name "Channel_4"}
	Channel_4 : Channel_460B8C40;
END_STRUCT
END_TYPE

// ---- DUTs/IO/Boxes/KL2641_8487B205.TcDUT
{attribute 'GeneratedUsingTerminal: KL2641'}
{attribute addProperty BoxType "KL2641"}
{attribute addProperty Description ""}
{attribute addProperty Physics ""}
{attribute addProperty Id "Channel_1AT %Q*Channel_2589C8DC0"}
{attribute addProperty CRC "2223485445"}
{attribute addProperty Size "0"}
TYPE KL2641_8487B205 :
STRUCT
	{attribute addProperty Name "Channel_1"}
	Channel_1 : Channel_2589C8DC;
END_STRUCT
END_TYPE

// ---- DUTs/IO/Boxes/KL_AF699C3C.TcDUT
{attribute 'GeneratedUsingTerminal: KL2641-0001'}
{attribute addProperty BoxType "KL2641-0001"}
{attribute addProperty Description ""}
{attribute addProperty Physics ""}
{attribute addProperty Id "Channel_1AT %Q*Channel_BF3661CD0"}
{attribute addProperty CRC "2942934076"}
{attribute addProperty Size "0"}
TYPE KL_AF699C3C :
STRUCT
	{attribute addProperty Name "Channel_1"}
	Channel_1 : Channel_BF3661CD;
END_STRUCT
END_TYPE

// ---- DUTs/IO/Boxes/KL2652_DCA75612.TcDUT
{attribute 'GeneratedUsingTerminal: KL2652'}
{attribute addProperty BoxType "KL2652"}
{attribute addProperty Description ""}
{attribute addProperty Physics ""}
{attribute addProperty Id "Channel_1AT %Q*Channel_460B8C400Channel_2AT %Q*Channel_460B8C400"}
{attribute addProperty CRC "3701954066"}
{attribute addProperty Size "0"}
TYPE KL2652_DCA75612 :
STRUCT
	{attribute addProperty Name "Channel_1"}
	Channel_1 : Channel_460B8C40;
	{attribute addProperty Name "Channel_2"}
	Channel_2 : Channel_460B8C40;
END_STRUCT
END_TYPE

// ---- DUTs/IO/Boxes/KL_6148C904.TcDUT
{attribute 'GeneratedUsingTerminal: KL2692-0001'}
{attribute addProperty BoxType "KL2692-0001"}
{attribute addProperty Description ""}
{attribute addProperty Physics ""}
{attribute addProperty Id "Channel_1AT %Q*Channel_6576A6810"}
{attribute addProperty CRC "1632160004"}
{attribute addProperty Size "0"}
TYPE KL_6148C904 :
STRUCT
	{attribute addProperty Name "Channel_1"}
	Channel_1 : Channel_6576A681;
END_STRUCT
END_TYPE

// ---- DUTs/IO/Boxes/KL2701_DE78D366.TcDUT
{attribute 'GeneratedUsingTerminal: KL2701'}
{attribute addProperty BoxType "KL2701"}
{attribute addProperty Description ""}
{attribute addProperty Physics ""}
{attribute addProperty Id "Channel_1AT %Q*Channel_460B8C400"}
{attribute addProperty CRC "3732460390"}
{attribute addProperty Size "0"}
TYPE KL2701_DE78D366 :
STRUCT
	{attribute addProperty Name "Channel_1"}
	Channel_1 : Channel_460B8C40;
END_STRUCT
END_TYPE

// ---- DUTs/IO/Boxes/KL2702_DCA75612.TcDUT
{attribute 'GeneratedUsingTerminal: KL2702'}
{attribute addProperty BoxType "KL2702"}
{attribute addProperty Description ""}
{attribute addProperty Physics ""}
{attribute addProperty Id "Channel_1AT %Q*Channel_460B8C400Channel_2AT %Q*Channel_460B8C400"}
{attribute addProperty CRC "3701954066"}
{attribute addProperty Size "0"}
TYPE KL2702_DCA75612 :
STRUCT
	{attribute addProperty Name "Channel_1"}
	Channel_1 : Channel_460B8C40;
	{attribute addProperty Name "Channel_2"}
	Channel_2 : Channel_460B8C40;
END_STRUCT
END_TYPE

// ---- DUTs/IO/Boxes/KL2712_DCA75612.TcDUT
{attribute 'GeneratedUsingTerminal: KL2712'}
{attribute addProperty BoxType "KL2712"}
{attribute addProperty Description ""}
{attribute addProperty Physics ""}
{attribute addProperty Id "Channel_1AT %Q*Channel_460B8C400Channel_2AT %Q*Channel_460B8C400"}
{attribute addProperty CRC "3701954066"}
{attribute addProperty Size "0"}
TYPE KL2712_DCA75612 :
STRUCT
	{attribute addProperty Name "Channel_1"}
	Channel_1 : Channel_460B8C40;
	{attribute addProperty Name "Channel_2"}
	Channel_2 : Channel_460B8C40;
END_STRUCT
END_TYPE

// ---- DUTs/IO/Boxes/KL2722_DCA75612.TcDUT
{attribute 'GeneratedUsingTerminal: KL2722'}
{attribute addProperty BoxType "KL2722"}
{attribute addProperty Description ""}
{attribute addProperty Physics ""}
{attribute addProperty Id "Channel_1AT %Q*Channel_460B8C400Channel_2AT %Q*Channel_460B8C400"}
{attribute addProperty CRC "3701954066"}
{attribute addProperty Size "0"}
TYPE KL2722_DCA75612 :
STRUCT
	{attribute addProperty Name "Channel_1"}
	Channel_1 : Channel_460B8C40;
	{attribute addProperty Name "Channel_2"}
	Channel_2 : Channel_460B8C40;
END_STRUCT
END_TYPE

// ---- DUTs/IO/Boxes/KL2732_DCA75612.TcDUT
{attribute 'GeneratedUsingTerminal: KL2732'}
{attribute addProperty BoxType "KL2732"}
{attribute addProperty Description ""}
{attribute addProperty Physics ""}
{attribute addProperty Id "Channel_1AT %Q*Channel_460B8C400Channel_2AT %Q*Channel_460B8C400"}
{attribute addProperty CRC "3701954066"}
{attribute addProperty Size "0"}
TYPE KL2732_DCA75612 :
STRUCT
	{attribute addProperty Name "Channel_1"}
	Channel_1 : Channel_460B8C40;
	{attribute addProperty Name "Channel_2"}
	Channel_2 : Channel_460B8C40;
END_STRUCT
END_TYPE

// ---- DUTs/IO/Boxes/KL2744_E49EE1EF.TcDUT
{attribute 'GeneratedUsingTerminal: KL2744'}
{attribute addProperty BoxType "KL2744"}
{attribute addProperty Description ""}
{attribute addProperty Physics ""}
{attribute addProperty Id "Channel_1AT %Q*Channel_460B8C400Channel_2AT %Q*Channel_460B8C400Channel_3AT %Q*Channel_460B8C400Channel_4AT %Q*Channel_460B8C400"}
{attribute addProperty CRC "3835617775"}
{attribute addProperty Size "0"}
TYPE KL2744_E49EE1EF :
STRUCT
	{attribute addProperty Name "Channel_1"}
	Channel_1 : Channel_460B8C40;
	{attribute addProperty Name "Channel_2"}
	Channel_2 : Channel_460B8C40;
	{attribute addProperty Name "Channel_3"}
	Channel_3 : Channel_460B8C40;
	{attribute addProperty Name "Channel_4"}
	Channel_4 : Channel_460B8C40;
END_STRUCT
END_TYPE

// ---- DUTs/IO/Boxes/KL2751_6148C904.TcDUT
{attribute 'GeneratedUsingTerminal: KL2751'}
{attribute addProperty BoxType "KL2751"}
{attribute addProperty Description ""}
{attribute addProperty Physics ""}
{attribute addProperty Id "Channel_1AT %Q*Channel_6576A6810"}
{attribute addProperty CRC "1632160004"}
{attribute addProperty Size "0"}
TYPE KL2751_6148C904 :
STRUCT
	{attribute addProperty Name "Channel_1"}
	Channel_1 : Channel_6576A681;
END_STRUCT
END_TYPE

// ---- DUTs/IO/Boxes/KL2761_6148C904.TcDUT
{attribute 'GeneratedUsingTerminal: KL2761'}
{attribute addProperty BoxType "KL2761"}
{attribute addProperty Description ""}
{attribute addProperty Physics ""}
{attribute addProperty Id "Channel_1AT %Q*Channel_6576A6810"}
{attribute addProperty CRC "1632160004"}
{attribute addProperty Size "0"}
TYPE KL2761_6148C904 :
STRUCT
	{attribute addProperty Name "Channel_1"}
	Channel_1 : Channel_6576A681;
END_STRUCT
END_TYPE

// ---- DUTs/IO/Boxes/KL2784_E49EE1EF.TcDUT
{attribute 'GeneratedUsingTerminal: KL2784'}
{attribute addProperty BoxType "KL2784"}
{attribute addProperty Description ""}
{attribute addProperty Physics ""}
{attribute addProperty Id "Channel_1AT %Q*Channel_460B8C400Channel_2AT %Q*Channel_460B8C400Channel_3AT %Q*Channel_460B8C400Channel_4AT %Q*Channel_460B8C400"}
{attribute addProperty CRC "3835617775"}
{attribute addProperty Size "0"}
TYPE KL2784_E49EE1EF :
STRUCT
	{attribute addProperty Name "Channel_1"}
	Channel_1 : Channel_460B8C40;
	{attribute addProperty Name "Channel_2"}
	Channel_2 : Channel_460B8C40;
	{attribute addProperty Name "Channel_3"}
	Channel_3 : Channel_460B8C40;
	{attribute addProperty Name "Channel_4"}
	Channel_4 : Channel_460B8C40;
END_STRUCT
END_TYPE

// ---- DUTs/IO/Boxes/KL2791_6148C904.TcDUT
{attribute 'GeneratedUsingTerminal: KL2791'}
{attribute addProperty BoxType "KL2791"}
{attribute addProperty Description ""}
{attribute addProperty Physics ""}
{attribute addProperty Id "Channel_1AT %Q*Channel_6576A6810"}
{attribute addProperty CRC "1632160004"}
{attribute addProperty Size "0"}
TYPE KL2791_6148C904 :
STRUCT
	{attribute addProperty Name "Channel_1"}
	Channel_1 : Channel_6576A681;
END_STRUCT
END_TYPE

// ---- DUTs/IO/Boxes/KL2794_E49EE1EF.TcDUT
{attribute 'GeneratedUsingTerminal: KL2794'}
{attribute addProperty BoxType "KL2794"}
{attribute addProperty Description ""}
{attribute addProperty Physics ""}
{attribute addProperty Id "Channel_1AT %Q*Channel_460B8C400Channel_2AT %Q*Channel_460B8C400Channel_3AT %Q*Channel_460B8C400Channel_4AT %Q*Channel_460B8C400"}
{attribute addProperty CRC "3835617775"}
{attribute addProperty Size "0"}
TYPE KL2794_E49EE1EF :
STRUCT
	{attribute addProperty Name "Channel_1"}
	Channel_1 : Channel_460B8C40;
	{attribute addProperty Name "Channel_2"}
	Channel_2 : Channel_460B8C40;
	{attribute addProperty Name "Channel_3"}
	Channel_3 : Channel_460B8C40;
	{attribute addProperty Name "Channel_4"}
	Channel_4 : Channel_460B8C40;
END_STRUCT
END_TYPE

// ---- DUTs/IO/Boxes/KL2798_CBAD53BF.TcDUT
{attribute 'GeneratedUsingTerminal: KL2798'}
{attribute addProperty BoxType "KL2798"}
{attribute addProperty Description ""}
{attribute addProperty Physics ""}
{attribute addProperty Id "Channel_1AT %Q*Channel_460B8C400Channel_2AT %Q*Channel_460B8C400Channel_3AT %Q*Channel_460B8C400Channel_4AT %Q*Channel_460B8C400Channel_5AT %Q*Channel_460B8C400Channel_6AT %Q*Channel_460B8C400Channel_7AT %Q*Channel_460B8C400Channel_8AT %Q*Channel_460B8C400"}
{attribute addProperty CRC "3417134015"}
{attribute addProperty Size "0"}
TYPE KL2798_CBAD53BF :
STRUCT
	{attribute addProperty Name "Channel_1"}
	Channel_1 : Channel_460B8C40;
	{attribute addProperty Name "Channel_2"}
	Channel_2 : Channel_460B8C40;
	{attribute addProperty Name "Channel_3"}
	Channel_3 : Channel_460B8C40;
	{attribute addProperty Name "Channel_4"}
	Channel_4 : Channel_460B8C40;
	{attribute addProperty Name "Channel_5"}
	Channel_5 : Channel_460B8C40;
	{attribute addProperty Name "Channel_6"}
	Channel_6 : Channel_460B8C40;
	{attribute addProperty Name "Channel_7"}
	Channel_7 : Channel_460B8C40;
	{attribute addProperty Name "Channel_8"}
	Channel_8 : Channel_460B8C40;
END_STRUCT
END_TYPE

// ---- DUTs/IO/Boxes/KL2808_CBAD53BF.TcDUT
{attribute 'GeneratedUsingTerminal: KL2808'}
{attribute addProperty BoxType "KL2808"}
{attribute addProperty Description ""}
{attribute addProperty Physics ""}
{attribute addProperty Id "Channel_1AT %Q*Channel_460B8C400Channel_2AT %Q*Channel_460B8C400Channel_3AT %Q*Channel_460B8C400Channel_4AT %Q*Channel_460B8C400Channel_5AT %Q*Channel_460B8C400Channel_6AT %Q*Channel_460B8C400Channel_7AT %Q*Channel_460B8C400Channel_8AT %Q*Channel_460B8C400"}
{attribute addProperty CRC "3417134015"}
{attribute addProperty Size "0"}
TYPE KL2808_CBAD53BF :
STRUCT
	{attribute addProperty Name "Channel_1"}
	Channel_1 : Channel_460B8C40;
	{attribute addProperty Name "Channel_2"}
	Channel_2 : Channel_460B8C40;
	{attribute addProperty Name "Channel_3"}
	Channel_3 : Channel_460B8C40;
	{attribute addProperty Name "Channel_4"}
	Channel_4 : Channel_460B8C40;
	{attribute addProperty Name "Channel_5"}
	Channel_5 : Channel_460B8C40;
	{attribute addProperty Name "Channel_6"}
	Channel_6 : Channel_460B8C40;
	{attribute addProperty Name "Channel_7"}
	Channel_7 : Channel_460B8C40;
	{attribute addProperty Name "Channel_8"}
	Channel_8 : Channel_460B8C40;
END_STRUCT
END_TYPE

// ---- DUTs/IO/Boxes/KL2819_28D63841.TcDUT
{attribute 'GeneratedUsingTerminal: KL2819'}
{attribute addProperty BoxType "KL2819"}
{attribute addProperty Description ""}
{attribute addProperty Physics ""}
{attribute addProperty Id "Channel_1AT %Q*Channel_2EC3E8CA0"}
{attribute addProperty CRC "685127745"}
{attribute addProperty Size "0"}
TYPE KL2819_28D63841 :
STRUCT
	{attribute addProperty Name "Channel_1"}
	Channel_1 : Channel_2EC3E8CA;
END_STRUCT
END_TYPE

// ---- DUTs/IO/Boxes/KL2828_CBAD53BF.TcDUT
{attribute 'GeneratedUsingTerminal: KL2828'}
{attribute addProperty BoxType "KL2828"}
{attribute addProperty Description ""}
{attribute addProperty Physics ""}
{attribute addProperty Id "Channel_1AT %Q*Channel_460B8C400Channel_2AT %Q*Channel_460B8C400Channel_3AT %Q*Channel_460B8C400Channel_4AT %Q*Channel_460B8C400Channel_5AT %Q*Channel_460B8C400Channel_6AT %Q*Channel_460B8C400Channel_7AT %Q*Channel_460B8C400Channel_8AT %Q*Channel_460B8C400"}
{attribute addProperty CRC "3417134015"}
{attribute addProperty Size "0"}
TYPE KL2828_CBAD53BF :
STRUCT
	{attribute addProperty Name "Channel_1"}
	Channel_1 : Channel_460B8C40;
	{attribute addProperty Name "Channel_2"}
	Channel_2 : Channel_460B8C40;
	{attribute addProperty Name "Channel_3"}
	Channel_3 : Channel_460B8C40;
	{attribute addProperty Name "Channel_4"}
	Channel_4 : Channel_460B8C40;
	{attribute addProperty Name "Channel_5"}
	Channel_5 : Channel_460B8C40;
	{attribute addProperty Name "Channel_6"}
	Channel_6 : Channel_460B8C40;
	{attribute addProperty Name "Channel_7"}
	Channel_7 : Channel_460B8C40;
	{attribute addProperty Name "Channel_8"}
	Channel_8 : Channel_460B8C40;
END_STRUCT
END_TYPE

// ---- DUTs/IO/Boxes/KL2809_F0D0C9F8.TcDUT
{attribute 'GeneratedUsingTerminal: KL2809'}
{attribute addProperty BoxType "KL2809"}
{attribute addProperty Description ""}
{attribute addProperty Physics ""}
{attribute addProperty Id "Channel_1AT %Q*Channel_460B8C400Channel_2AT %Q*Channel_460B8C400Channel_3AT %Q*Channel_460B8C400Channel_4AT %Q*Channel_460B8C400Channel_5AT %Q*Channel_460B8C400Channel_6AT %Q*Channel_460B8C400Channel_7AT %Q*Channel_460B8C400Channel_8AT %Q*Channel_460B8C400Channel_9AT %Q*Channel_460B8C400Channel_10AT %Q*Channel_460B8C400Channel_11AT %Q*Channel_460B8C400Channel_12AT %Q*Channel_460B8C400Channel_13AT %Q*Channel_460B8C400Channel_14AT %Q*Channel_460B8C400Channel_15AT %Q*Channel_460B8C400Channel_16AT %Q*Channel_460B8C400"}
{attribute addProperty CRC "4040215032"}
{attribute addProperty Size "0"}
TYPE KL2809_F0D0C9F8 :
STRUCT
	{attribute addProperty Name "Channel_1"}
	Channel_1 : Channel_460B8C40;
	{attribute addProperty Name "Channel_2"}
	Channel_2 : Channel_460B8C40;
	{attribute addProperty Name "Channel_3"}
	Channel_3 : Channel_460B8C40;
	{attribute addProperty Name "Channel_4"}
	Channel_4 : Channel_460B8C40;
	{attribute addProperty Name "Channel_5"}
	Channel_5 : Channel_460B8C40;
	{attribute addProperty Name "Channel_6"}
	Channel_6 : Channel_460B8C40;
	{attribute addProperty Name "Channel_7"}
	Channel_7 : Channel_460B8C40;
	{attribute addProperty Name "Channel_8"}
	Channel_8 : Channel_460B8C40;
	{attribute addProperty Name "Channel_9"}
	Channel_9 : Channel_460B8C40;
	{attribute addProperty Name "Channel_10"}
	Channel_10 : Channel_460B8C40;
	{attribute addProperty Name "Channel_11"}
	Channel_11 : Channel_460B8C40;
	{attribute addProperty Name "Channel_12"}
	Channel_12 : Channel_460B8C40;
	{attribute addProperty Name "Channel_13"}
	Channel_13 : Channel_460B8C40;
	{attribute addProperty Name "Channel_14"}
	Channel_14 : Channel_460B8C40;
	{attribute addProperty Name "Channel_15"}
	Channel_15 : Channel_460B8C40;
	{attribute addProperty Name "Channel_16"}
	Channel_16 : Channel_460B8C40;
END_STRUCT
END_TYPE

// ---- DUTs/IO/Boxes/KL2872_F0D0C9F8.TcDUT
{attribute 'GeneratedUsingTerminal: KL2872'}
{attribute addProperty BoxType "KL2872"}
{attribute addProperty Description ""}
{attribute addProperty Physics ""}
{attribute addProperty Id "Channel_1AT %Q*Channel_460B8C400Channel_2AT %Q*Channel_460B8C400Channel_3AT %Q*Channel_460B8C400Channel_4AT %Q*Channel_460B8C400Channel_5AT %Q*Channel_460B8C400Channel_6AT %Q*Channel_460B8C400Channel_7AT %Q*Channel_460B8C400Channel_8AT %Q*Channel_460B8C400Channel_9AT %Q*Channel_460B8C400Channel_10AT %Q*Channel_460B8C400Channel_11AT %Q*Channel_460B8C400Channel_12AT %Q*Channel_460B8C400Channel_13AT %Q*Channel_460B8C400Channel_14AT %Q*Channel_460B8C400Channel_15AT %Q*Channel_460B8C400Channel_16AT %Q*Channel_460B8C400"}
{attribute addProperty CRC "4040215032"}
{attribute addProperty Size "0"}
TYPE KL2872_F0D0C9F8 :
STRUCT
	{attribute addProperty Name "Channel_1"}
	Channel_1 : Channel_460B8C40;
	{attribute addProperty Name "Channel_2"}
	Channel_2 : Channel_460B8C40;
	{attribute addProperty Name "Channel_3"}
	Channel_3 : Channel_460B8C40;
	{attribute addProperty Name "Channel_4"}
	Channel_4 : Channel_460B8C40;
	{attribute addProperty Name "Channel_5"}
	Channel_5 : Channel_460B8C40;
	{attribute addProperty Name "Channel_6"}
	Channel_6 : Channel_460B8C40;
	{attribute addProperty Name "Channel_7"}
	Channel_7 : Channel_460B8C40;
	{attribute addProperty Name "Channel_8"}
	Channel_8 : Channel_460B8C40;
	{attribute addProperty Name "Channel_9"}
	Channel_9 : Channel_460B8C40;
	{attribute addProperty Name "Channel_10"}
	Channel_10 : Channel_460B8C40;
	{attribute addProperty Name "Channel_11"}
	Channel_11 : Channel_460B8C40;
	{attribute addProperty Name "Channel_12"}
	Channel_12 : Channel_460B8C40;
	{attribute addProperty Name "Channel_13"}
	Channel_13 : Channel_460B8C40;
	{attribute addProperty Name "Channel_14"}
	Channel_14 : Channel_460B8C40;
	{attribute addProperty Name "Channel_15"}
	Channel_15 : Channel_460B8C40;
	{attribute addProperty Name "Channel_16"}
	Channel_16 : Channel_460B8C40;
END_STRUCT
END_TYPE

// ---- DUTs/IO/Boxes/KL2889_F0D0C9F8.TcDUT
{attribute 'GeneratedUsingTerminal: KL2889'}
{attribute addProperty BoxType "KL2889"}
{attribute addProperty Description ""}
{attribute addProperty Physics ""}
{attribute addProperty Id "Channel_1AT %Q*Channel_460B8C400Channel_2AT %Q*Channel_460B8C400Channel_3AT %Q*Channel_460B8C400Channel_4AT %Q*Channel_460B8C400Channel_5AT %Q*Channel_460B8C400Channel_6AT %Q*Channel_460B8C400Channel_7AT %Q*Channel_460B8C400Channel_8AT %Q*Channel_460B8C400Channel_9AT %Q*Channel_460B8C400Channel_10AT %Q*Channel_460B8C400Channel_11AT %Q*Channel_460B8C400Channel_12AT %Q*Channel_460B8C400Channel_13AT %Q*Channel_460B8C400Channel_14AT %Q*Channel_460B8C400Channel_15AT %Q*Channel_460B8C400Channel_16AT %Q*Channel_460B8C400"}
{attribute addProperty CRC "4040215032"}
{attribute addProperty Size "0"}
TYPE KL2889_F0D0C9F8 :
STRUCT
	{attribute addProperty Name "Channel_1"}
	Channel_1 : Channel_460B8C40;
	{attribute addProperty Name "Channel_2"}
	Channel_2 : Channel_460B8C40;
	{attribute addProperty Name "Channel_3"}
	Channel_3 : Channel_460B8C40;
	{attribute addProperty Name "Channel_4"}
	Channel_4 : Channel_460B8C40;
	{attribute addProperty Name "Channel_5"}
	Channel_5 : Channel_460B8C40;
	{attribute addProperty Name "Channel_6"}
	Channel_6 : Channel_460B8C40;
	{attribute addProperty Name "Channel_7"}
	Channel_7 : Channel_460B8C40;
	{attribute addProperty Name "Channel_8"}
	Channel_8 : Channel_460B8C40;
	{attribute addProperty Name "Channel_9"}
	Channel_9 : Channel_460B8C40;
	{attribute addProperty Name "Channel_10"}
	Channel_10 : Channel_460B8C40;
	{attribute addProperty Name "Channel_11"}
	Channel_11 : Channel_460B8C40;
	{attribute addProperty Name "Channel_12"}
	Channel_12 : Channel_460B8C40;
	{attribute addProperty Name "Channel_13"}
	Channel_13 : Channel_460B8C40;
	{attribute addProperty Name "Channel_14"}
	Channel_14 : Channel_460B8C40;
	{attribute addProperty Name "Channel_15"}
	Channel_15 : Channel_460B8C40;
	{attribute addProperty Name "Channel_16"}
	Channel_16 : Channel_460B8C40;
END_STRUCT
END_TYPE

// ---- DUTs/IO/Boxes/KL2904_7F0D69A9.TcDUT
{attribute 'GeneratedUsingTerminal: KL2904'}
{attribute addProperty BoxType "KL2904"}
{attribute addProperty Description ""}
{attribute addProperty Physics ""}
{attribute addProperty Id "Channel_1AT %Q*Channel_1D6668A90"}
{attribute addProperty CRC "2131585449"}
{attribute addProperty Size "0"}
TYPE KL2904_7F0D69A9 :
STRUCT
	{attribute addProperty Name "Channel_1"}
	Channel_1 : Channel_1D6668A9;
END_STRUCT
END_TYPE

// ---- DUTs/IO/Boxes/KL_F0D0C9F8.TcDUT
{attribute 'GeneratedUsingTerminal: KL2002-0050'}
{attribute addProperty BoxType "KL2002-0050"}
{attribute addProperty Description ""}
{attribute addProperty Physics ""}
{attribute addProperty Id "Channel_1AT %Q*Channel_460B8C400Channel_2AT %Q*Channel_460B8C400Channel_3AT %Q*Channel_460B8C400Channel_4AT %Q*Channel_460B8C400Channel_5AT %Q*Channel_460B8C400Channel_6AT %Q*Channel_460B8C400Channel_7AT %Q*Channel_460B8C400Channel_8AT %Q*Channel_460B8C400Channel_9AT %Q*Channel_460B8C400Channel_10AT %Q*Channel_460B8C400Channel_11AT %Q*Channel_460B8C400Channel_12AT %Q*Channel_460B8C400Channel_13AT %Q*Channel_460B8C400Channel_14AT %Q*Channel_460B8C400Channel_15AT %Q*Channel_460B8C400Channel_16AT %Q*Channel_460B8C400"}
{attribute addProperty CRC "4040215032"}
{attribute addProperty Size "0"}
TYPE KL_F0D0C9F8 :
STRUCT
	{attribute addProperty Name "Channel_1"}
	Channel_1 : Channel_460B8C40;
	{attribute addProperty Name "Channel_2"}
	Channel_2 : Channel_460B8C40;
	{attribute addProperty Name "Channel_3"}
	Channel_3 : Channel_460B8C40;
	{attribute addProperty Name "Channel_4"}
	Channel_4 : Channel_460B8C40;
	{attribute addProperty Name "Channel_5"}
	Channel_5 : Channel_460B8C40;
	{attribute addProperty Name "Channel_6"}
	Channel_6 : Channel_460B8C40;
	{attribute addProperty Name "Channel_7"}
	Channel_7 : Channel_460B8C40;
	{attribute addProperty Name "Channel_8"}
	Channel_8 : Channel_460B8C40;
	{attribute addProperty Name "Channel_9"}
	Channel_9 : Channel_460B8C40;
	{attribute addProperty Name "Channel_10"}
	Channel_10 : Channel_460B8C40;
	{attribute addProperty Name "Channel_11"}
	Channel_11 : Channel_460B8C40;
	{attribute addProperty Name "Channel_12"}
	Channel_12 : Channel_460B8C40;
	{attribute addProperty Name "Channel_13"}
	Channel_13 : Channel_460B8C40;
	{attribute addProperty Name "Channel_14"}
	Channel_14 : Channel_460B8C40;
	{attribute addProperty Name "Channel_15"}
	Channel_15 : Channel_460B8C40;
	{attribute addProperty Name "Channel_16"}
	Channel_16 : Channel_460B8C40;
END_STRUCT
END_TYPE

// ---- DUTs/IO/Boxes/KL_CF002DCA.TcDUT
{attribute 'GeneratedUsingTerminal: KL2004-0050'}
{attribute addProperty BoxType "KL2004-0050"}
{attribute addProperty Description ""}
{attribute addProperty Physics ""}
{attribute addProperty Id "Channel_1AT %Q*Channel_460B8C400Channel_2AT %Q*Channel_460B8C400Channel_3AT %Q*Channel_460B8C400Channel_4AT %Q*Channel_460B8C400Channel_5AT %Q*Channel_460B8C400Channel_6AT %Q*Channel_460B8C400Channel_7AT %Q*Channel_460B8C400Channel_8AT %Q*Channel_460B8C400Channel_9AT %Q*Channel_460B8C400Channel_10AT %Q*Channel_460B8C400Channel_11AT %Q*Channel_460B8C400Channel_12AT %Q*Channel_460B8C400Channel_13AT %Q*Channel_460B8C400Channel_14AT %Q*Channel_460B8C400Channel_15AT %Q*Channel_460B8C400Channel_16AT %Q*Channel_460B8C400Channel_17AT %Q*Channel_460B8C400Channel_18AT %Q*Channel_460B8C400Channel_19AT %Q*Channel_460B8C400Channel_20AT %Q*Channel_460B8C400Channel_21AT %Q*Channel_460B8C400Channel_22AT %Q*Channel_460B8C400Channel_23AT %Q*Channel_460B8C400Channel_24AT %Q*Channel_460B8C400Channel_25AT %Q*Channel_460B8C400Channel_26AT %Q*Channel_460B8C400Channel_27AT %Q*Channel_460B8C400Channel_28AT %Q*Channel_460B8C400Channel_29AT %Q*Channel_460B8C400Channel_30AT %Q*Channel_460B8C400Channel_31AT %Q*Channel_460B8C400Channel_32AT %Q*Channel_460B8C400"}
{attribute addProperty CRC "3472895434"}
{attribute addProperty Size "0"}
TYPE KL_CF002DCA :
STRUCT
	{attribute addProperty Name "Channel_1"}
	Channel_1 : Channel_460B8C40;
	{attribute addProperty Name "Channel_2"}
	Channel_2 : Channel_460B8C40;
	{attribute addProperty Name "Channel_3"}
	Channel_3 : Channel_460B8C40;
	{attribute addProperty Name "Channel_4"}
	Channel_4 : Channel_460B8C40;
	{attribute addProperty Name "Channel_5"}
	Channel_5 : Channel_460B8C40;
	{attribute addProperty Name "Channel_6"}
	Channel_6 : Channel_460B8C40;
	{attribute addProperty Name "Channel_7"}
	Channel_7 : Channel_460B8C40;
	{attribute addProperty Name "Channel_8"}
	Channel_8 : Channel_460B8C40;
	{attribute addProperty Name "Channel_9"}
	Channel_9 : Channel_460B8C40;
	{attribute addProperty Name "Channel_10"}
	Channel_10 : Channel_460B8C40;
	{attribute addProperty Name "Channel_11"}
	Channel_11 : Channel_460B8C40;
	{attribute addProperty Name "Channel_12"}
	Channel_12 : Channel_460B8C40;
	{attribute addProperty Name "Channel_13"}
	Channel_13 : Channel_460B8C40;
	{attribute addProperty Name "Channel_14"}
	Channel_14 : Channel_460B8C40;
	{attribute addProperty Name "Channel_15"}
	Channel_15 : Channel_460B8C40;
	{attribute addProperty Name "Channel_16"}
	Channel_16 : Channel_460B8C40;
	{attribute addProperty Name "Channel_17"}
	Channel_17 : Channel_460B8C40;
	{attribute addProperty Name "Channel_18"}
	Channel_18 : Channel_460B8C40;
	{attribute addProperty Name "Channel_19"}
	Channel_19 : Channel_460B8C40;
	{attribute addProperty Name "Channel_20"}
	Channel_20 : Channel_460B8C40;
	{attribute addProperty Name "Channel_21"}
	Channel_21 : Channel_460B8C40;
	{attribute addProperty Name "Channel_22"}
	Channel_22 : Channel_460B8C40;
	{attribute addProperty Name "Channel_23"}
	Channel_23 : Channel_460B8C40;
	{attribute addProperty Name "Channel_24"}
	Channel_24 : Channel_460B8C40;
	{attribute addProperty Name "Channel_25"}
	Channel_25 : Channel_460B8C40;
	{attribute addProperty Name "Channel_26"}
	Channel_26 : Channel_460B8C40;
	{attribute addProperty Name "Channel_27"}
	Channel_27 : Channel_460B8C40;
	{attribute addProperty Name "Channel_28"}
	Channel_28 : Channel_460B8C40;
	{attribute addProperty Name "Channel_29"}
	Channel_29 : Channel_460B8C40;
	{attribute addProperty Name "Channel_30"}
	Channel_30 : Channel_460B8C40;
	{attribute addProperty Name "Channel_31"}
	Channel_31 : Channel_460B8C40;
	{attribute addProperty Name "Channel_32"}
	Channel_32 : Channel_460B8C40;
END_STRUCT
END_TYPE

// ---- DUTs/IO/Boxes/KL_F7A5EEBF.TcDUT
{attribute 'GeneratedUsingTerminal: KL2008-0050'}
{attribute addProperty BoxType "KL2008-0050"}
{attribute addProperty Description ""}
{attribute addProperty Physics ""}
{attribute addProperty Id "Channel_1AT %Q*Channel_460B8C400Channel_2AT %Q*Channel_460B8C400Channel_3AT %Q*Channel_460B8C400Channel_4AT %Q*Channel_460B8C400Channel_5AT %Q*Channel_460B8C400Channel_6AT %Q*Channel_460B8C400Channel_7AT %Q*Channel_460B8C400Channel_8AT %Q*Channel_460B8C400Channel_9AT %Q*Channel_460B8C400Channel_10AT %Q*Channel_460B8C400Channel_11AT %Q*Channel_460B8C400Channel_12AT %Q*Channel_460B8C400Channel_13AT %Q*Channel_460B8C400Channel_14AT %Q*Channel_460B8C400Channel_15AT %Q*Channel_460B8C400Channel_16AT %Q*Channel_460B8C400Channel_17AT %Q*Channel_460B8C400Channel_18AT %Q*Channel_460B8C400Channel_19AT %Q*Channel_460B8C400Channel_20AT %Q*Channel_460B8C400Channel_21AT %Q*Channel_460B8C400Channel_22AT %Q*Channel_460B8C400Channel_23AT %Q*Channel_460B8C400Channel_24AT %Q*Channel_460B8C400Channel_25AT %Q*Channel_460B8C400Channel_26AT %Q*Channel_460B8C400Channel_27AT %Q*Channel_460B8C400Channel_28AT %Q*Channel_460B8C400Channel_29AT %Q*Channel_460B8C400Channel_30AT %Q*Channel_460B8C400Channel_31AT %Q*Channel_460B8C400Channel_32AT %Q*Channel_460B8C400Channel_33AT %Q*Channel_460B8C400Channel_34AT %Q*Channel_460B8C400Channel_35AT %Q*Channel_460B8C400Channel_36AT %Q*Channel_460B8C400Channel_37AT %Q*Channel_460B8C400Channel_38AT %Q*Channel_460B8C400Channel_39AT %Q*Channel_460B8C400Channel_40AT %Q*Channel_460B8C400Channel_41AT %Q*Channel_460B8C400Channel_42AT %Q*Channel_460B8C400Channel_43AT %Q*Channel_460B8C400Channel_44AT %Q*Channel_460B8C400Channel_45AT %Q*Channel_460B8C400Channel_46AT %Q*Channel_460B8C400Channel_47AT %Q*Channel_460B8C400Channel_48AT %Q*Channel_460B8C400Channel_49AT %Q*Channel_460B8C400Channel_50AT %Q*Channel_460B8C400Channel_51AT %Q*Channel_460B8C400Channel_52AT %Q*Channel_460B8C400Channel_53AT %Q*Channel_460B8C400Channel_54AT %Q*Channel_460B8C400Channel_55AT %Q*Channel_460B8C400Channel_56AT %Q*Channel_460B8C400Channel_57AT %Q*Channel_460B8C400Channel_58AT %Q*Channel_460B8C400Channel_59AT %Q*Channel_460B8C400Channel_60AT %Q*Channel_460B8C400Channel_61AT %Q*Channel_460B8C400Channel_62AT %Q*Channel_460B8C400Channel_63AT %Q*Channel_460B8C400Channel_64AT %Q*Channel_460B8C400"}
{attribute addProperty CRC "4154846911"}
{attribute addProperty Size "0"}
TYPE KL_F7A5EEBF :
STRUCT
	{attribute addProperty Name "Channel_1"}
	Channel_1 : Channel_460B8C40;
	{attribute addProperty Name "Channel_2"}
	Channel_2 : Channel_460B8C40;
	{attribute addProperty Name "Channel_3"}
	Channel_3 : Channel_460B8C40;
	{attribute addProperty Name "Channel_4"}
	Channel_4 : Channel_460B8C40;
	{attribute addProperty Name "Channel_5"}
	Channel_5 : Channel_460B8C40;
	{attribute addProperty Name "Channel_6"}
	Channel_6 : Channel_460B8C40;
	{attribute addProperty Name "Channel_7"}
	Channel_7 : Channel_460B8C40;
	{attribute addProperty Name "Channel_8"}
	Channel_8 : Channel_460B8C40;
	{attribute addProperty Name "Channel_9"}
	Channel_9 : Channel_460B8C40;
	{attribute addProperty Name "Channel_10"}
	Channel_10 : Channel_460B8C40;
	{attribute addProperty Name "Channel_11"}
	Channel_11 : Channel_460B8C40;
	{attribute addProperty Name "Channel_12"}
	Channel_12 : Channel_460B8C40;
	{attribute addProperty Name "Channel_13"}
	Channel_13 : Channel_460B8C40;
	{attribute addProperty Name "Channel_14"}
	Channel_14 : Channel_460B8C40;
	{attribute addProperty Name "Channel_15"}
	Channel_15 : Channel_460B8C40;
	{attribute addProperty Name "Channel_16"}
	Channel_16 : Channel_460B8C40;
	{attribute addProperty Name "Channel_17"}
	Channel_17 : Channel_460B8C40;
	{attribute addProperty Name "Channel_18"}
	Channel_18 : Channel_460B8C40;
	{attribute addProperty Name "Channel_19"}
	Channel_19 : Channel_460B8C40;
	{attribute addProperty Name "Channel_20"}
	Channel_20 : Channel_460B8C40;
	{attribute addProperty Name "Channel_21"}
	Channel_21 : Channel_460B8C40;
	{attribute addProperty Name "Channel_22"}
	Channel_22 : Channel_460B8C40;
	{attribute addProperty Name "Channel_23"}
	Channel_23 : Channel_460B8C40;
	{attribute addProperty Name "Channel_24"}
	Channel_24 : Channel_460B8C40;
	{attribute addProperty Name "Channel_25"}
	Channel_25 : Channel_460B8C40;
	{attribute addProperty Name "Channel_26"}
	Channel_26 : Channel_460B8C40;
	{attribute addProperty Name "Channel_27"}
	Channel_27 : Channel_460B8C40;
	{attribute addProperty Name "Channel_28"}
	Channel_28 : Channel_460B8C40;
	{attribute addProperty Name "Channel_29"}
	Channel_29 : Channel_460B8C40;
	{attribute addProperty Name "Channel_30"}
	Channel_30 : Channel_460B8C40;
	{attribute addProperty Name "Channel_31"}
	Channel_31 : Channel_460B8C40;
	{attribute addProperty Name "Channel_32"}
	Channel_32 : Channel_460B8C40;
	{attribute addProperty Name "Channel_33"}
	Channel_33 : Channel_460B8C40;
	{attribute addProperty Name "Channel_34"}
	Channel_34 : Channel_460B8C40;
	{attribute addProperty Name "Channel_35"}
	Channel_35 : Channel_460B8C40;
	{attribute addProperty Name "Channel_36"}
	Channel_36 : Channel_460B8C40;
	{attribute addProperty Name "Channel_37"}
	Channel_37 : Channel_460B8C40;
	{attribute addProperty Name "Channel_38"}
	Channel_38 : Channel_460B8C40;
	{attribute addProperty Name "Channel_39"}
	Channel_39 : Channel_460B8C40;
	{attribute addProperty Name "Channel_40"}
	Channel_40 : Channel_460B8C40;
	{attribute addProperty Name "Channel_41"}
	Channel_41 : Channel_460B8C40;
	{attribute addProperty Name "Channel_42"}
	Channel_42 : Channel_460B8C40;
	{attribute addProperty Name "Channel_43"}
	Channel_43 : Channel_460B8C40;
	{attribute addProperty Name "Channel_44"}
	Channel_44 : Channel_460B8C40;
	{attribute addProperty Name "Channel_45"}
	Channel_45 : Channel_460B8C40;
	{attribute addProperty Name "Channel_46"}
	Channel_46 : Channel_460B8C40;
	{attribute addProperty Name "Channel_47"}
	Channel_47 : Channel_460B8C40;
	{attribute addProperty Name "Channel_48"}
	Channel_48 : Channel_460B8C40;
	{attribute addProperty Name "Channel_49"}
	Channel_49 : Channel_460B8C40;
	{attribute addProperty Name "Channel_50"}
	Channel_50 : Channel_460B8C40;
	{attribute addProperty Name "Channel_51"}
	Channel_51 : Channel_460B8C40;
	{attribute addProperty Name "Channel_52"}
	Channel_52 : Channel_460B8C40;
	{attribute addProperty Name "Channel_53"}
	Channel_53 : Channel_460B8C40;
	{attribute addProperty Name "Channel_54"}
	Channel_54 : Channel_460B8C40;
	{attribute addProperty Name "Channel_55"}
	Channel_55 : Channel_460B8C40;
	{attribute addProperty Name "Channel_56"}
	Channel_56 : Channel_460B8C40;
	{attribute addProperty Name "Channel_57"}
	Channel_57 : Channel_460B8C40;
	{attribute addProperty Name "Channel_58"}
	Channel_58 : Channel_460B8C40;
	{attribute addProperty Name "Channel_59"}
	Channel_59 : Channel_460B8C40;
	{attribute addProperty Name "Channel_60"}
	Channel_60 : Channel_460B8C40;
	{attribute addProperty Name "Channel_61"}
	Channel_61 : Channel_460B8C40;
	{attribute addProperty Name "Channel_62"}
	Channel_62 : Channel_460B8C40;
	{attribute addProperty Name "Channel_63"}
	Channel_63 : Channel_460B8C40;
	{attribute addProperty Name "Channel_64"}
	Channel_64 : Channel_460B8C40;
END_STRUCT
END_TYPE

// ---- DUTs/IO/Boxes/KL_E49EE1EF.TcDUT
{attribute 'GeneratedUsingTerminal: KL2604-0050'}
{attribute addProperty BoxType "KL2604-0050"}
{attribute addProperty Description ""}
{attribute addProperty Physics ""}
{attribute addProperty Id "Channel_1AT %Q*Channel_460B8C400Channel_2AT %Q*Channel_460B8C400Channel_3AT %Q*Channel_460B8C400Channel_4AT %Q*Channel_460B8C400"}
{attribute addProperty CRC "3835617775"}
{attribute addProperty Size "0"}
TYPE KL_E49EE1EF :
STRUCT
	{attribute addProperty Name "Channel_1"}
	Channel_1 : Channel_460B8C40;
	{attribute addProperty Name "Channel_2"}
	Channel_2 : Channel_460B8C40;
	{attribute addProperty Name "Channel_3"}
	Channel_3 : Channel_460B8C40;
	{attribute addProperty Name "Channel_4"}
	Channel_4 : Channel_460B8C40;
END_STRUCT
END_TYPE

// ---- DUTs/IO/Boxes/KL_F206FFFF.TcDUT
{attribute 'GeneratedUsingTerminal: KL2642-0050'}
{attribute addProperty BoxType "KL2642-0050"}
{attribute addProperty Description ""}
{attribute addProperty Physics ""}
{attribute addProperty Id "Channel_1AT %Q*Channel_F5DB8AD10Channel_2AT %Q*Channel_F5DB8AD10"}
{attribute addProperty CRC "4060545023"}
{attribute addProperty Size "0"}
TYPE KL_F206FFFF :
STRUCT
	{attribute addProperty Name "Channel_1"}
	Channel_1 : Channel_F5DB8AD1;
	{attribute addProperty Name "Channel_2"}
	Channel_2 : Channel_F5DB8AD1;
END_STRUCT
END_TYPE

// ---- DUTs/IO/Boxes/KL_13ED1AE5.TcDUT
{attribute 'GeneratedUsingTerminal: KL2652-0050'}
{attribute addProperty BoxType "KL2652-0050"}
{attribute addProperty Description ""}
{attribute addProperty Physics ""}
{attribute addProperty Id "Channel_1AT %Q*Channel_6D8B740B0Channel_2AT %Q*Channel_6D8B740B0"}
{attribute addProperty CRC "334306021"}
{attribute addProperty Size "0"}
TYPE KL_13ED1AE5 :
STRUCT
	{attribute addProperty Name "Channel_1"}
	Channel_1 : Channel_6D8B740B;
	{attribute addProperty Name "Channel_2"}
	Channel_2 : Channel_6D8B740B;
END_STRUCT
END_TYPE

// ---- DUTs/IO/Boxes/KL2774_6148C904.TcDUT
{attribute 'GeneratedUsingTerminal: KL2774'}
{attribute addProperty BoxType "KL2774"}
{attribute addProperty Description ""}
{attribute addProperty Physics ""}
{attribute addProperty Id "Channel_1AT %Q*Channel_6576A6810"}
{attribute addProperty CRC "1632160004"}
{attribute addProperty Size "0"}
TYPE KL2774_6148C904 :
STRUCT
	{attribute addProperty Name "Channel_1"}
	Channel_1 : Channel_6576A681;
END_STRUCT
END_TYPE

// ---- DUTs/IO/Boxes/KL_CBAD53BF.TcDUT
{attribute 'GeneratedUsingTerminal: KL2018-0020'}
{attribute addProperty BoxType "KL2018-0020"}
{attribute addProperty Description ""}
{attribute addProperty Physics ""}
{attribute addProperty Id "Channel_1AT %Q*Channel_460B8C400Channel_2AT %Q*Channel_460B8C400Channel_3AT %Q*Channel_460B8C400Channel_4AT %Q*Channel_460B8C400Channel_5AT %Q*Channel_460B8C400Channel_6AT %Q*Channel_460B8C400Channel_7AT %Q*Channel_460B8C400Channel_8AT %Q*Channel_460B8C400"}
{attribute addProperty CRC "3417134015"}
{attribute addProperty Size "0"}
TYPE KL_CBAD53BF :
STRUCT
	{attribute addProperty Name "Channel_1"}
	Channel_1 : Channel_460B8C40;
	{attribute addProperty Name "Channel_2"}
	Channel_2 : Channel_460B8C40;
	{attribute addProperty Name "Channel_3"}
	Channel_3 : Channel_460B8C40;
	{attribute addProperty Name "Channel_4"}
	Channel_4 : Channel_460B8C40;
	{attribute addProperty Name "Channel_5"}
	Channel_5 : Channel_460B8C40;
	{attribute addProperty Name "Channel_6"}
	Channel_6 : Channel_460B8C40;
	{attribute addProperty Name "Channel_7"}
	Channel_7 : Channel_460B8C40;
	{attribute addProperty Name "Channel_8"}
	Channel_8 : Channel_460B8C40;
END_STRUCT
END_TYPE

// ---- DUTs/IO/Boxes/KL3001_6148C904.TcDUT
{attribute 'GeneratedUsingTerminal: KL3001'}
{attribute addProperty BoxType "KL3001"}
{attribute addProperty Description ""}
{attribute addProperty Physics ""}
{attribute addProperty Id "Channel_1AT %Q*Channel_6576A6810"}
{attribute addProperty CRC "1632160004"}
{attribute addProperty Size "0"}
TYPE KL3001_6148C904 :
STRUCT
	{attribute addProperty Name "Channel_1"}
	Channel_1 : Channel_6576A681;
END_STRUCT
END_TYPE

// ---- DUTs/IO/Boxes/KL3002_B0461874.TcDUT
{attribute 'GeneratedUsingTerminal: KL3002'}
{attribute addProperty BoxType "KL3002"}
{attribute addProperty Description ""}
{attribute addProperty Physics ""}
{attribute addProperty Id "Channel_1AT %Q*Channel_6576A6810Channel_2AT %Q*Channel_6576A6810"}
{attribute addProperty CRC "2957383796"}
{attribute addProperty Size "0"}
TYPE KL3002_B0461874 :
STRUCT
	{attribute addProperty Name "Channel_1"}
	Channel_1 : Channel_6576A681;
	{attribute addProperty Name "Channel_2"}
	Channel_2 : Channel_6576A681;
END_STRUCT
END_TYPE

// ---- DUTs/IO/Boxes/KL3011_6148C904.TcDUT
{attribute 'GeneratedUsingTerminal: KL3011'}
{attribute addProperty BoxType "KL3011"}
{attribute addProperty Description ""}
{attribute addProperty Physics ""}
{attribute addProperty Id "Channel_1AT %Q*Channel_6576A6810"}
{attribute addProperty CRC "1632160004"}
{attribute addProperty Size "0"}
TYPE KL3011_6148C904 :
STRUCT
	{attribute addProperty Name "Channel_1"}
	Channel_1 : Channel_6576A681;
END_STRUCT
END_TYPE

// ---- DUTs/IO/Boxes/KL3012_B0461874.TcDUT
{attribute 'GeneratedUsingTerminal: KL3012'}
{attribute addProperty BoxType "KL3012"}
{attribute addProperty Description ""}
{attribute addProperty Physics ""}
{attribute addProperty Id "Channel_1AT %Q*Channel_6576A6810Channel_2AT %Q*Channel_6576A6810"}
{attribute addProperty CRC "2957383796"}
{attribute addProperty Size "0"}
TYPE KL3012_B0461874 :
STRUCT
	{attribute addProperty Name "Channel_1"}
	Channel_1 : Channel_6576A681;
	{attribute addProperty Name "Channel_2"}
	Channel_2 : Channel_6576A681;
END_STRUCT
END_TYPE

// ---- DUTs/IO/Boxes/KL3021_6148C904.TcDUT
{attribute 'GeneratedUsingTerminal: KL3021'}
{attribute addProperty BoxType "KL3021"}
{attribute addProperty Description ""}
{attribute addProperty Physics ""}
{attribute addProperty Id "Channel_1AT %Q*Channel_6576A6810"}
{attribute addProperty CRC "1632160004"}
{attribute addProperty Size "0"}
TYPE KL3021_6148C904 :
STRUCT
	{attribute addProperty Name "Channel_1"}
	Channel_1 : Channel_6576A681;
END_STRUCT
END_TYPE

// ---- DUTs/IO/Boxes/KL3022_B0461874.TcDUT
{attribute 'GeneratedUsingTerminal: KL3022'}
{attribute addProperty BoxType "KL3022"}
{attribute addProperty Description ""}
{attribute addProperty Physics ""}
{attribute addProperty Id "Channel_1AT %Q*Channel_6576A6810Channel_2AT %Q*Channel_6576A6810"}
{attribute addProperty CRC "2957383796"}
{attribute addProperty Size "0"}
TYPE KL3022_B0461874 :
STRUCT
	{attribute addProperty Name "Channel_1"}
	Channel_1 : Channel_6576A681;
	{attribute addProperty Name "Channel_2"}
	Channel_2 : Channel_6576A681;
END_STRUCT
END_TYPE

// ---- DUTs/IO/Boxes/KL3041_6148C904.TcDUT
{attribute 'GeneratedUsingTerminal: KL3041'}
{attribute addProperty BoxType "KL3041"}
{attribute addProperty Description ""}
{attribute addProperty Physics ""}
{attribute addProperty Id "Channel_1AT %Q*Channel_6576A6810"}
{attribute addProperty CRC "1632160004"}
{attribute addProperty Size "0"}
TYPE KL3041_6148C904 :
STRUCT
	{attribute addProperty Name "Channel_1"}
	Channel_1 : Channel_6576A681;
END_STRUCT
END_TYPE

// ---- DUTs/IO/Boxes/KL3042_B0461874.TcDUT
{attribute 'GeneratedUsingTerminal: KL3042'}
{attribute addProperty BoxType "KL3042"}
{attribute addProperty Description ""}
{attribute addProperty Physics ""}
{attribute addProperty Id "Channel_1AT %Q*Channel_6576A6810Channel_2AT %Q*Channel_6576A6810"}
{attribute addProperty CRC "2957383796"}
{attribute addProperty Size "0"}
TYPE KL3042_B0461874 :
STRUCT
	{attribute addProperty Name "Channel_1"}
	Channel_1 : Channel_6576A681;
	{attribute addProperty Name "Channel_2"}
	Channel_2 : Channel_6576A681;
END_STRUCT
END_TYPE

// ---- DUTs/IO/Boxes/KL3044_8BE38B75.TcDUT
{attribute 'GeneratedUsingTerminal: KL3044'}
{attribute addProperty BoxType "KL3044"}
{attribute addProperty Description ""}
{attribute addProperty Physics ""}
{attribute addProperty Id "Channel_1AT %Q*Channel_6576A6810Channel_2AT %Q*Channel_6576A6810Channel_3AT %Q*Channel_6576A6810Channel_4AT %Q*Channel_6576A6810"}
{attribute addProperty CRC "2346945397"}
{attribute addProperty Size "0"}
TYPE KL3044_8BE38B75 :
STRUCT
	{attribute addProperty Name "Channel_1"}
	Channel_1 : Channel_6576A681;
	{attribute addProperty Name "Channel_2"}
	Channel_2 : Channel_6576A681;
	{attribute addProperty Name "Channel_3"}
	Channel_3 : Channel_6576A681;
	{attribute addProperty Name "Channel_4"}
	Channel_4 : Channel_6576A681;
END_STRUCT
END_TYPE

// ---- DUTs/IO/Boxes/KL_ACD69469.TcDUT
{attribute 'GeneratedUsingTerminal: KL3044-0001'}
{attribute addProperty BoxType "KL3044-0001"}
{attribute addProperty Description ""}
{attribute addProperty Physics ""}
{attribute addProperty Id "Channel_1AT %I*0Channel_2AT %I*0Channel_3AT %I*0Channel_4AT %I*0"}
{attribute addProperty CRC "2899743849"}
{attribute addProperty Size "0"}
TYPE KL_ACD69469 :
STRUCT
	{attribute addProperty Name "Channel_1"}
	Channel_1 : ;
	{attribute addProperty Name "Channel_2"}
	Channel_2 : ;
	{attribute addProperty Name "Channel_3"}
	Channel_3 : ;
	{attribute addProperty Name "Channel_4"}
	Channel_4 : ;
END_STRUCT
END_TYPE

// ---- DUTs/IO/Boxes/KL3051_6148C904.TcDUT
{attribute 'GeneratedUsingTerminal: KL3051'}
{attribute addProperty BoxType "KL3051"}
{attribute addProperty Description ""}
{attribute addProperty Physics ""}
{attribute addProperty Id "Channel_1AT %Q*Channel_6576A6810"}
{attribute addProperty CRC "1632160004"}
{attribute addProperty Size "0"}
TYPE KL3051_6148C904 :
STRUCT
	{attribute addProperty Name "Channel_1"}
	Channel_1 : Channel_6576A681;
END_STRUCT
END_TYPE

// ---- DUTs/IO/Boxes/KL3052_B0461874.TcDUT
{attribute 'GeneratedUsingTerminal: KL3052'}
{attribute addProperty BoxType "KL3052"}
{attribute addProperty Description ""}
{attribute addProperty Physics ""}
{attribute addProperty Id "Channel_1AT %Q*Channel_6576A6810Channel_2AT %Q*Channel_6576A6810"}
{attribute addProperty CRC "2957383796"}
{attribute addProperty Size "0"}
TYPE KL3052_B0461874 :
STRUCT
	{attribute addProperty Name "Channel_1"}
	Channel_1 : Channel_6576A681;
	{attribute addProperty Name "Channel_2"}
	Channel_2 : Channel_6576A681;
END_STRUCT
END_TYPE

// ---- DUTs/IO/Boxes/KL3054_8BE38B75.TcDUT
{attribute 'GeneratedUsingTerminal: KL3054'}
{attribute addProperty BoxType "KL3054"}
{attribute addProperty Description ""}
{attribute addProperty Physics ""}
{attribute addProperty Id "Channel_1AT %Q*Channel_6576A6810Channel_2AT %Q*Channel_6576A6810Channel_3AT %Q*Channel_6576A6810Channel_4AT %Q*Channel_6576A6810"}
{attribute addProperty CRC "2346945397"}
{attribute addProperty Size "0"}
TYPE KL3054_8BE38B75 :
STRUCT
	{attribute addProperty Name "Channel_1"}
	Channel_1 : Channel_6576A681;
	{attribute addProperty Name "Channel_2"}
	Channel_2 : Channel_6576A681;
	{attribute addProperty Name "Channel_3"}
	Channel_3 : Channel_6576A681;
	{attribute addProperty Name "Channel_4"}
	Channel_4 : Channel_6576A681;
END_STRUCT
END_TYPE

// ---- DUTs/IO/Boxes/KL3061_6148C904.TcDUT
{attribute 'GeneratedUsingTerminal: KL3061'}
{attribute addProperty BoxType "KL3061"}
{attribute addProperty Description ""}
{attribute addProperty Physics ""}
{attribute addProperty Id "Channel_1AT %Q*Channel_6576A6810"}
{attribute addProperty CRC "1632160004"}
{attribute addProperty Size "0"}
TYPE KL3061_6148C904 :
STRUCT
	{attribute addProperty Name "Channel_1"}
	Channel_1 : Channel_6576A681;
END_STRUCT
END_TYPE

// ---- DUTs/IO/Boxes/KL3062_B0461874.TcDUT
{attribute 'GeneratedUsingTerminal: KL3062'}
{attribute addProperty BoxType "KL3062"}
{attribute addProperty Description ""}
{attribute addProperty Physics ""}
{attribute addProperty Id "Channel_1AT %Q*Channel_6576A6810Channel_2AT %Q*Channel_6576A6810"}
{attribute addProperty CRC "2957383796"}
{attribute addProperty Size "0"}
TYPE KL3062_B0461874 :
STRUCT
	{attribute addProperty Name "Channel_1"}
	Channel_1 : Channel_6576A681;
	{attribute addProperty Name "Channel_2"}
	Channel_2 : Channel_6576A681;
END_STRUCT
END_TYPE

// ---- DUTs/IO/Boxes/KL3064_8BE38B75.TcDUT
{attribute 'GeneratedUsingTerminal: KL3064'}
{attribute addProperty BoxType "KL3064"}
{attribute addProperty Description ""}
{attribute addProperty Physics ""}
{attribute addProperty Id "Channel_1AT %Q*Channel_6576A6810Channel_2AT %Q*Channel_6576A6810Channel_3AT %Q*Channel_6576A6810Channel_4AT %Q*Channel_6576A6810"}
{attribute addProperty CRC "2346945397"}
{attribute addProperty Size "0"}
TYPE KL3064_8BE38B75 :
STRUCT
	{attribute addProperty Name "Channel_1"}
	Channel_1 : Channel_6576A681;
	{attribute addProperty Name "Channel_2"}
	Channel_2 : Channel_6576A681;
	{attribute addProperty Name "Channel_3"}
	Channel_3 : Channel_6576A681;
	{attribute addProperty Name "Channel_4"}
	Channel_4 : Channel_6576A681;
END_STRUCT
END_TYPE

// ---- DUTs/IO/Boxes/KL3102_B0461874.TcDUT
{attribute 'GeneratedUsingTerminal: KL3102'}
{attribute addProperty BoxType "KL3102"}
{attribute addProperty Description ""}
{attribute addProperty Physics ""}
{attribute addProperty Id "Channel_1AT %Q*Channel_6576A6810Channel_2AT %Q*Channel_6576A6810"}
{attribute addProperty CRC "2957383796"}
{attribute addProperty Size "0"}
TYPE KL3102_B0461874 :
STRUCT
	{attribute addProperty Name "Channel_1"}
	Channel_1 : Channel_6576A681;
	{attribute addProperty Name "Channel_2"}
	Channel_2 : Channel_6576A681;
END_STRUCT
END_TYPE

// ---- DUTs/IO/Boxes/KL3112_B0461874.TcDUT
{attribute 'GeneratedUsingTerminal: KL3112'}
{attribute addProperty BoxType "KL3112"}
{attribute addProperty Description ""}
{attribute addProperty Physics ""}
{attribute addProperty Id "Channel_1AT %Q*Channel_6576A6810Channel_2AT %Q*Channel_6576A6810"}
{attribute addProperty CRC "2957383796"}
{attribute addProperty Size "0"}
TYPE KL3112_B0461874 :
STRUCT
	{attribute addProperty Name "Channel_1"}
	Channel_1 : Channel_6576A681;
	{attribute addProperty Name "Channel_2"}
	Channel_2 : Channel_6576A681;
END_STRUCT
END_TYPE

// ---- DUTs/IO/Boxes/KL3122_B0461874.TcDUT
{attribute 'GeneratedUsingTerminal: KL3122'}
{attribute addProperty BoxType "KL3122"}
{attribute addProperty Description ""}
{attribute addProperty Physics ""}
{attribute addProperty Id "Channel_1AT %Q*Channel_6576A6810Channel_2AT %Q*Channel_6576A6810"}
{attribute addProperty CRC "2957383796"}
{attribute addProperty Size "0"}
TYPE KL3122_B0461874 :
STRUCT
	{attribute addProperty Name "Channel_1"}
	Channel_1 : Channel_6576A681;
	{attribute addProperty Name "Channel_2"}
	Channel_2 : Channel_6576A681;
END_STRUCT
END_TYPE

// ---- DUTs/IO/Boxes/KL3132_B0461874.TcDUT
{attribute 'GeneratedUsingTerminal: KL3132'}
{attribute addProperty BoxType "KL3132"}
{attribute addProperty Description ""}
{attribute addProperty Physics ""}
{attribute addProperty Id "Channel_1AT %Q*Channel_6576A6810Channel_2AT %Q*Channel_6576A6810"}
{attribute addProperty CRC "2957383796"}
{attribute addProperty Size "0"}
TYPE KL3132_B0461874 :
STRUCT
	{attribute addProperty Name "Channel_1"}
	Channel_1 : Channel_6576A681;
	{attribute addProperty Name "Channel_2"}
	Channel_2 : Channel_6576A681;
END_STRUCT
END_TYPE

// ---- DUTs/IO/Boxes/KL3142_78388DBB.TcDUT
{attribute 'GeneratedUsingTerminal: KL3142'}
{attribute addProperty BoxType "KL3142"}
{attribute addProperty Description ""}
{attribute addProperty Physics ""}
{attribute addProperty Id "Channel_1AT %Q*Channel_03CEAA5E0Channel_2AT %Q*Channel_03CEAA5E0"}
{attribute addProperty CRC "2016972219"}
{attribute addProperty Size "0"}
TYPE KL3142_78388DBB :
STRUCT
	{attribute addProperty Name "Channel_1"}
	Channel_1 : Channel_03CEAA5E;
	{attribute addProperty Name "Channel_2"}
	Channel_2 : Channel_03CEAA5E;
END_STRUCT
END_TYPE

// ---- DUTs/IO/Boxes/KL3152_78388DBB.TcDUT
{attribute 'GeneratedUsingTerminal: KL3152'}
{attribute addProperty BoxType "KL3152"}
{attribute addProperty Description ""}
{attribute addProperty Physics ""}
{attribute addProperty Id "Channel_1AT %Q*Channel_03CEAA5E0Channel_2AT %Q*Channel_03CEAA5E0"}
{attribute addProperty CRC "2016972219"}
{attribute addProperty Size "0"}
TYPE KL3152_78388DBB :
STRUCT
	{attribute addProperty Name "Channel_1"}
	Channel_1 : Channel_03CEAA5E;
	{attribute addProperty Name "Channel_2"}
	Channel_2 : Channel_03CEAA5E;
END_STRUCT
END_TYPE

// ---- DUTs/IO/Boxes/KL3158_8BE38B75.TcDUT
{attribute 'GeneratedUsingTerminal: KL3158'}
{attribute addProperty BoxType "KL3158"}
{attribute addProperty Description ""}
{attribute addProperty Physics ""}
{attribute addProperty Id "Channel_1AT %Q*Channel_6576A6810Channel_2AT %Q*Channel_6576A6810Channel_3AT %Q*Channel_6576A6810Channel_4AT %Q*Channel_6576A6810"}
{attribute addProperty CRC "2346945397"}
{attribute addProperty Size "0"}
TYPE KL3158_8BE38B75 :
STRUCT
	{attribute addProperty Name "Channel_1"}
	Channel_1 : Channel_6576A681;
	{attribute addProperty Name "Channel_2"}
	Channel_2 : Channel_6576A681;
	{attribute addProperty Name "Channel_3"}
	Channel_3 : Channel_6576A681;
	{attribute addProperty Name "Channel_4"}
	Channel_4 : Channel_6576A681;
END_STRUCT
END_TYPE

// ---- DUTs/IO/Boxes/KL3162_78388DBB.TcDUT
{attribute 'GeneratedUsingTerminal: KL3162'}
{attribute addProperty BoxType "KL3162"}
{attribute addProperty Description ""}
{attribute addProperty Physics ""}
{attribute addProperty Id "Channel_1AT %Q*Channel_03CEAA5E0Channel_2AT %Q*Channel_03CEAA5E0"}
{attribute addProperty CRC "2016972219"}
{attribute addProperty Size "0"}
TYPE KL3162_78388DBB :
STRUCT
	{attribute addProperty Name "Channel_1"}
	Channel_1 : Channel_03CEAA5E;
	{attribute addProperty Name "Channel_2"}
	Channel_2 : Channel_03CEAA5E;
END_STRUCT
END_TYPE

// ---- DUTs/IO/Boxes/KL3172_78388DBB.TcDUT
{attribute 'GeneratedUsingTerminal: KL3172'}
{attribute addProperty BoxType "KL3172"}
{attribute addProperty Description ""}
{attribute addProperty Physics ""}
{attribute addProperty Id "Channel_1AT %Q*Channel_03CEAA5E0Channel_2AT %Q*Channel_03CEAA5E0"}
{attribute addProperty CRC "2016972219"}
{attribute addProperty Size "0"}
TYPE KL3172_78388DBB :
STRUCT
	{attribute addProperty Name "Channel_1"}
	Channel_1 : Channel_03CEAA5E;
	{attribute addProperty Name "Channel_2"}
	Channel_2 : Channel_03CEAA5E;
END_STRUCT
END_TYPE

// ---- DUTs/IO/Boxes/KL_78388DBB.TcDUT
{attribute 'GeneratedUsingTerminal: KL3172-0002'}
{attribute addProperty BoxType "KL3172-0002"}
{attribute addProperty Description ""}
{attribute addProperty Physics ""}
{attribute addProperty Id "Channel_1AT %Q*Channel_03CEAA5E0Channel_2AT %Q*Channel_03CEAA5E0"}
{attribute addProperty CRC "2016972219"}
{attribute addProperty Size "0"}
TYPE KL_78388DBB :
STRUCT
	{attribute addProperty Name "Channel_1"}
	Channel_1 : Channel_03CEAA5E;
	{attribute addProperty Name "Channel_2"}
	Channel_2 : Channel_03CEAA5E;
END_STRUCT
END_TYPE

// ---- DUTs/IO/Boxes/KL3182_B0461874.TcDUT
{attribute 'GeneratedUsingTerminal: KL3182'}
{attribute addProperty BoxType "KL3182"}
{attribute addProperty Description ""}
{attribute addProperty Physics ""}
{attribute addProperty Id "Channel_1AT %Q*Channel_6576A6810Channel_2AT %Q*Channel_6576A6810"}
{attribute addProperty CRC "2957383796"}
{attribute addProperty Size "0"}
TYPE KL3182_B0461874 :
STRUCT
	{attribute addProperty Name "Channel_1"}
	Channel_1 : Channel_6576A681;
	{attribute addProperty Name "Channel_2"}
	Channel_2 : Channel_6576A681;
END_STRUCT
END_TYPE

// ---- DUTs/IO/Boxes/KL3201_6148C904.TcDUT
{attribute 'GeneratedUsingTerminal: KL3201'}
{attribute addProperty BoxType "KL3201"}
{attribute addProperty Description ""}
{attribute addProperty Physics ""}
{attribute addProperty Id "Channel_1AT %Q*Channel_6576A6810"}
{attribute addProperty CRC "1632160004"}
{attribute addProperty Size "0"}
TYPE KL3201_6148C904 :
STRUCT
	{attribute addProperty Name "Channel_1"}
	Channel_1 : Channel_6576A681;
END_STRUCT
END_TYPE

// ---- DUTs/IO/Boxes/KL3202_B0461874.TcDUT
{attribute 'GeneratedUsingTerminal: KL3202'}
{attribute addProperty BoxType "KL3202"}
{attribute addProperty Description ""}
{attribute addProperty Physics ""}
{attribute addProperty Id "Channel_1AT %Q*Channel_6576A6810Channel_2AT %Q*Channel_6576A6810"}
{attribute addProperty CRC "2957383796"}
{attribute addProperty Size "0"}
TYPE KL3202_B0461874 :
STRUCT
	{attribute addProperty Name "Channel_1"}
	Channel_1 : Channel_6576A681;
	{attribute addProperty Name "Channel_2"}
	Channel_2 : Channel_6576A681;
END_STRUCT
END_TYPE

// ---- DUTs/IO/Boxes/KL3204_8BE38B75.TcDUT
{attribute 'GeneratedUsingTerminal: KL3204'}
{attribute addProperty BoxType "KL3204"}
{attribute addProperty Description ""}
{attribute addProperty Physics ""}
{attribute addProperty Id "Channel_1AT %Q*Channel_6576A6810Channel_2AT %Q*Channel_6576A6810Channel_3AT %Q*Channel_6576A6810Channel_4AT %Q*Channel_6576A6810"}
{attribute addProperty CRC "2346945397"}
{attribute addProperty Size "0"}
TYPE KL3204_8BE38B75 :
STRUCT
	{attribute addProperty Name "Channel_1"}
	Channel_1 : Channel_6576A681;
	{attribute addProperty Name "Channel_2"}
	Channel_2 : Channel_6576A681;
	{attribute addProperty Name "Channel_3"}
	Channel_3 : Channel_6576A681;
	{attribute addProperty Name "Channel_4"}
	Channel_4 : Channel_6576A681;
END_STRUCT
END_TYPE

// ---- DUTs/IO/Boxes/KL_8BE38B75.TcDUT
{attribute 'GeneratedUsingTerminal: KL3208-0002'}
{attribute addProperty BoxType "KL3208-0002"}
{attribute addProperty Description ""}
{attribute addProperty Physics ""}
{attribute addProperty Id "Channel_1AT %Q*Channel_6576A6810Channel_2AT %Q*Channel_6576A6810Channel_3AT %Q*Channel_6576A6810Channel_4AT %Q*Channel_6576A6810"}
{attribute addProperty CRC "2346945397"}
{attribute addProperty Size "0"}
TYPE KL_8BE38B75 :
STRUCT
	{attribute addProperty Name "Channel_1"}
	Channel_1 : Channel_6576A681;
	{attribute addProperty Name "Channel_2"}
	Channel_2 : Channel_6576A681;
	{attribute addProperty Name "Channel_3"}
	Channel_3 : Channel_6576A681;
	{attribute addProperty Name "Channel_4"}
	Channel_4 : Channel_6576A681;
END_STRUCT
END_TYPE

// ---- DUTs/IO/Boxes/KL3214_8BE38B75.TcDUT
{attribute 'GeneratedUsingTerminal: KL3214'}
{attribute addProperty BoxType "KL3214"}
{attribute addProperty Description ""}
{attribute addProperty Physics ""}
{attribute addProperty Id "Channel_1AT %Q*Channel_6576A6810Channel_2AT %Q*Channel_6576A6810Channel_3AT %Q*Channel_6576A6810Channel_4AT %Q*Channel_6576A6810"}
{attribute addProperty CRC "2346945397"}
{attribute addProperty Size "0"}
TYPE KL3214_8BE38B75 :
STRUCT
	{attribute addProperty Name "Channel_1"}
	Channel_1 : Channel_6576A681;
	{attribute addProperty Name "Channel_2"}
	Channel_2 : Channel_6576A681;
	{attribute addProperty Name "Channel_3"}
	Channel_3 : Channel_6576A681;
	{attribute addProperty Name "Channel_4"}
	Channel_4 : Channel_6576A681;
END_STRUCT
END_TYPE

// ---- DUTs/IO/Boxes/KL3222_B0461874.TcDUT
{attribute 'GeneratedUsingTerminal: KL3222'}
{attribute addProperty BoxType "KL3222"}
{attribute addProperty Description ""}
{attribute addProperty Physics ""}
{attribute addProperty Id "Channel_1AT %Q*Channel_6576A6810Channel_2AT %Q*Channel_6576A6810"}
{attribute addProperty CRC "2957383796"}
{attribute addProperty Size "0"}
TYPE KL3222_B0461874 :
STRUCT
	{attribute addProperty Name "Channel_1"}
	Channel_1 : Channel_6576A681;
	{attribute addProperty Name "Channel_2"}
	Channel_2 : Channel_6576A681;
END_STRUCT
END_TYPE

// ---- DUTs/IO/Boxes/KL3224_8BE38B75.TcDUT
{attribute 'GeneratedUsingTerminal: KL3224'}
{attribute addProperty BoxType "KL3224"}
{attribute addProperty Description ""}
{attribute addProperty Physics ""}
{attribute addProperty Id "Channel_1AT %Q*Channel_6576A6810Channel_2AT %Q*Channel_6576A6810Channel_3AT %Q*Channel_6576A6810Channel_4AT %Q*Channel_6576A6810"}
{attribute addProperty CRC "2346945397"}
{attribute addProperty Size "0"}
TYPE KL3224_8BE38B75 :
STRUCT
	{attribute addProperty Name "Channel_1"}
	Channel_1 : Channel_6576A681;
	{attribute addProperty Name "Channel_2"}
	Channel_2 : Channel_6576A681;
	{attribute addProperty Name "Channel_3"}
	Channel_3 : Channel_6576A681;
	{attribute addProperty Name "Channel_4"}
	Channel_4 : Channel_6576A681;
END_STRUCT
END_TYPE

// ---- DUTs/IO/Boxes/KL3228_8BE38B75.TcDUT
{attribute 'GeneratedUsingTerminal: KL3228'}
{attribute addProperty BoxType "KL3228"}
{attribute addProperty Description ""}
{attribute addProperty Physics ""}
{attribute addProperty Id "Channel_1AT %Q*Channel_6576A6810Channel_2AT %Q*Channel_6576A6810Channel_3AT %Q*Channel_6576A6810Channel_4AT %Q*Channel_6576A6810"}
{attribute addProperty CRC "2346945397"}
{attribute addProperty Size "0"}
TYPE KL3228_8BE38B75 :
STRUCT
	{attribute addProperty Name "Channel_1"}
	Channel_1 : Channel_6576A681;
	{attribute addProperty Name "Channel_2"}
	Channel_2 : Channel_6576A681;
	{attribute addProperty Name "Channel_3"}
	Channel_3 : Channel_6576A681;
	{attribute addProperty Name "Channel_4"}
	Channel_4 : Channel_6576A681;
END_STRUCT
END_TYPE

// ---- DUTs/IO/Boxes/KL3302_B0461874.TcDUT
{attribute 'GeneratedUsingTerminal: KL3302'}
{attribute addProperty BoxType "KL3302"}
{attribute addProperty Description ""}
{attribute addProperty Physics ""}
{attribute addProperty Id "Channel_1AT %Q*Channel_6576A6810Channel_2AT %Q*Channel_6576A6810"}
{attribute addProperty CRC "2957383796"}
{attribute addProperty Size "0"}
TYPE KL3302_B0461874 :
STRUCT
	{attribute addProperty Name "Channel_1"}
	Channel_1 : Channel_6576A681;
	{attribute addProperty Name "Channel_2"}
	Channel_2 : Channel_6576A681;
END_STRUCT
END_TYPE

// ---- DUTs/IO/Boxes/KL3311_6148C904.TcDUT
{attribute 'GeneratedUsingTerminal: KL3311'}
{attribute addProperty BoxType "KL3311"}
{attribute addProperty Description ""}
{attribute addProperty Physics ""}
{attribute addProperty Id "Channel_1AT %Q*Channel_6576A6810"}
{attribute addProperty CRC "1632160004"}
{attribute addProperty Size "0"}
TYPE KL3311_6148C904 :
STRUCT
	{attribute addProperty Name "Channel_1"}
	Channel_1 : Channel_6576A681;
END_STRUCT
END_TYPE

// ---- DUTs/IO/Boxes/KL3312_B0461874.TcDUT
{attribute 'GeneratedUsingTerminal: KL3312'}
{attribute addProperty BoxType "KL3312"}
{attribute addProperty Description ""}
{attribute addProperty Physics ""}
{attribute addProperty Id "Channel_1AT %Q*Channel_6576A6810Channel_2AT %Q*Channel_6576A6810"}
{attribute addProperty CRC "2957383796"}
{attribute addProperty Size "0"}
TYPE KL3312_B0461874 :
STRUCT
	{attribute addProperty Name "Channel_1"}
	Channel_1 : Channel_6576A681;
	{attribute addProperty Name "Channel_2"}
	Channel_2 : Channel_6576A681;
END_STRUCT
END_TYPE

// ---- DUTs/IO/Boxes/KL3314_8BE38B75.TcDUT
{attribute 'GeneratedUsingTerminal: KL3314'}
{attribute addProperty BoxType "KL3314"}
{attribute addProperty Description ""}
{attribute addProperty Physics ""}
{attribute addProperty Id "Channel_1AT %Q*Channel_6576A6810Channel_2AT %Q*Channel_6576A6810Channel_3AT %Q*Channel_6576A6810Channel_4AT %Q*Channel_6576A6810"}
{attribute addProperty CRC "2346945397"}
{attribute addProperty Size "0"}
TYPE KL3314_8BE38B75 :
STRUCT
	{attribute addProperty Name "Channel_1"}
	Channel_1 : Channel_6576A681;
	{attribute addProperty Name "Channel_2"}
	Channel_2 : Channel_6576A681;
	{attribute addProperty Name "Channel_3"}
	Channel_3 : Channel_6576A681;
	{attribute addProperty Name "Channel_4"}
	Channel_4 : Channel_6576A681;
END_STRUCT
END_TYPE

// ---- DUTs/IO/Boxes/KL3351_33637CB0.TcDUT
{attribute 'GeneratedUsingTerminal: KL3351'}
{attribute addProperty BoxType "KL3351"}
{attribute addProperty Description ""}
{attribute addProperty Physics ""}
{attribute addProperty Id "Channel_1AT %Q*Channel_2DA3FF3C0"}
{attribute addProperty CRC "862158000"}
{attribute addProperty Size "0"}
TYPE KL3351_33637CB0 :
STRUCT
	{attribute addProperty Name "Channel_1"}
	Channel_1 : Channel_2DA3FF3C;
END_STRUCT
END_TYPE

